3552:L P[2314]  R[157] mm/sec CNT100 Offset,PR[24:Rotate_Offset] ;
3553:L P[2315]  R[157] mm/sec CNT100 Offset,PR[24:Rotate_Offset] ;
3554:L P[2316]  R[157] mm/sec CNT100 Offset,PR[24:Rotate_Offset] ;
3555:L P[2317]  R[157] mm/sec CNT100 Offset,PR[24:Rotate_Offset] ;
3556: !Pass176 ;
3557: LBL[1176:Pass176] ;
3558:L P[2318]  R[157] mm/sec FINE Offset,PR[78:Offst_apprch]  ;
3559: WAIT   0.20(sec) ;
3560:L P[2318]  R[157] mm/sec CNT100 TA    0.00sec,CALL RUN_LASER_START Offset,PR[25:Start_Offset] ;
3562:L P[2319]  R[157] mm/sec CNT100 Offset,PR[24:Rotate_Offset] ;
3563:L P[2320]  R[157] mm/sec CNT100 Offset,PR[24:Rotate_Offset] ;
3564:L P[2321]  R[157] mm/sec CNT100 Offset,PR[24:Rotate_Offset] ;
3565:L P[2322]  R[157] mm/sec CNT100 TA    0.00sec,CALL RUN_LASER_STOP Offset,PR[26:Stop_Offset] ;
3567:L P[2322]  R[157] mm/sec FINE Offset,PR[76:Offst_dprt] ;
3568:L P[2323]  R[157] mm/sec CNT100 Offset,PR[24:Rotate_Offset] ;
3569:L P[2324]  R[157] mm/sec CNT100 Offset,PR[24:Rotate_Offset] ;
3570:L P[2325]  R[157] mm/sec CNT100 Offset,PR[24:Rotate_Offset] ;
3571:L P[2326]  R[157] mm/sec CNT100 Offset,PR[24:Rotate_Offset] ;
3572:L P[2327]  R[157] mm/sec CNT100 Offset,PR[24:Rotate_Offset] ;
3573:L P[2328]  R[157] mm/sec CNT100 Offset,PR[24:Rotate_Offset] ;
3574: !Pass177 ;
3575: LBL[1177:Pass177] ;
3576:L P[2329]  R[157] mm/sec FINE Offset,PR[78:Offst_apprch]  ;
3577: WAIT   0.20(sec) ;
3578:L P[2329]  R[157] mm/sec CNT100 TA    0.00sec,CALL RUN_LASER_START Offset,PR[25:Start_Offset] ;
3580:L P[2330]  R[157] mm/sec CNT100 Offset,PR[24:Rotate_Offset] ;
3581:L P[2331]  R[157] mm/sec CNT100 Offset,PR[24:Rotate_Offset] ;
3582:L P[2332]  R[157] mm/sec CNT100 Offset,PR[24:Rotate_Offset] ;
3583:L P[2333]  R[157] mm/sec CNT100 TA    0.00sec,CALL RUN_LASER_STOP Offset,PR[26:Stop_Offset] ;
3585:L P[2333]  R[157] mm/sec FINE Offset,PR[76:Offst_dprt] ;
3586:L P[2334]  R[157] mm/sec CNT100 Offset,PR[24:Rotate_Offset] ;
3587:L P[2335]  R[157] mm/sec CNT100 Offset,PR[24:Rotate_Offset] ;
3588:L P[2336]  R[157] mm/sec CNT100 Offset,PR[24:Rotate_Offset] ;
3589:L P[2337]  R[157] mm/sec CNT100 Offset,PR[24:Rotate_Offset] ;
3590:L P[2338]  R[157] mm/sec CNT100 Offset,PR[24:Rotate_Offset] ;
3591:L P[2339]  R[157] mm/sec CNT100 Offset,PR[24:Rotate_Offset] ;
3592: !Pass178 ;
3593: LBL[1178:Pass178] ;
3594:L P[2340]  R[157] mm/sec FINE Offset,PR[78:Offst_apprch]  ;
3595: WAIT   0.20(sec) ;
3596:L P[2340]  R[157] mm/sec CNT100 TA    0.00sec,CALL RUN_LASER_START Offset,PR[25:Start_Offset] ;
3598:L P[2341]  R[157] mm/sec CNT100 Offset,PR[24:Rotate_Offset] ;
3599:L P[2342]  R[157] mm/sec CNT100 Offset,PR[24:Rotate_Offset] ;
3600:L P[2343]  R[157] mm/sec CNT100 Offset,PR[24:Rotate_Offset] ;
3601:L P[2344]  R[157] mm/sec CNT100 TA    0.00sec,CALL RUN_LASER_STOP Offset,PR[26:Stop_Offset] ;
3603:L P[2344]  R[157] mm/sec FINE Offset,PR[76:Offst_dprt] ;
3604:L P[2345]  R[157] mm/sec CNT100 Offset,PR[24:Rotate_Offset] ;
3605:L P[2346]  R[157] mm/sec CNT100 Offset,PR[24:Rotate_Offset] ;
3606:L P[2347]  R[157] mm/sec CNT100 Offset,PR[24:Rotate_Offset] ;
3607:L P[2348]  R[157] mm/sec CNT100 Offset,PR[24:Rotate_Offset] ;
3608:L P[2349]  R[157] mm/sec CNT100 Offset,PR[24:Rotate_Offset] ;
3609:L P[2350]  R[157] mm/sec CNT100 Offset,PR[24:Rotate_Offset] ;
3610: !Pass179 ;
3611: LBL[1179:Pass179] ;
3612:L P[2351]  R[157] mm/sec FINE Offset,PR[78:Offst_apprch]  ;
3613: WAIT   0.20(sec) ;
3614:L P[2351]  R[157] mm/sec CNT100 TA    0.00sec,CALL RUN_LASER_START Offset,PR[25:Start_Offset] ;
3616:L P[2352]  R[157] mm/sec CNT100 Offset,PR[24:Rotate_Offset] ;
3617:L P[2353]  R[157] mm/sec CNT100 TA    0.00sec,CALL RUN_LASER_STOP Offset,PR[26:Stop_Offset] ;
3619:L P[2353]  R[157] mm/sec FINE Offset,PR[76:Offst_dprt] ;
3620:L P[2354]  R[157] mm/sec CNT100 Offset,PR[24:Rotate_Offset] ;
3621:L P[2355]  R[157] mm/sec CNT100 Offset,PR[24:Rotate_Offset] ;
3622:L P[2356]  R[157] mm/sec CNT100 Offset,PR[24:Rotate_Offset] ;
3623:L P[2357]  R[157] mm/sec CNT100 Offset,PR[24:Rotate_Offset] ;
3624:L P[2358]  R[157] mm/sec CNT100 Offset,PR[24:Rotate_Offset] ;
3625:L P[2359]  R[157] mm/sec CNT100 Offset,PR[24:Rotate_Offset] ;
3626: !Pass180 ;
3627: LBL[1180:Pass180] ;
3628:L P[2360]  R[157] mm/sec FINE Offset,PR[78:Offst_apprch]  ;
3629: WAIT   0.20(sec) ;
3630:L P[2360]  R[157] mm/sec CNT100 TA    0.00sec,CALL RUN_LASER_START Offset,PR[25:Start_Offset] ;
3632:L P[2361]  R[157] mm/sec CNT100 Offset,PR[24:Rotate_Offset] ;
3633:L P[2362]  R[157] mm/sec CNT100 TA    0.00sec,CALL RUN_LASER_STOP Offset,PR[26:Stop_Offset] ;
3635:L P[2362]  R[157] mm/sec FINE Offset,PR[76:Offst_dprt] ;
3636:L P[2363]  R[157] mm/sec CNT100 Offset,PR[24:Rotate_Offset] ;
3637:L P[2364]  R[157] mm/sec CNT100 Offset,PR[24:Rotate_Offset] ;
3638:L P[2365]  R[157] mm/sec CNT100 Offset,PR[24:Rotate_Offset] ;
3639:L P[2366]  R[157] mm/sec CNT100 Offset,PR[24:Rotate_Offset] ;
3640:L P[2367]  R[157] mm/sec CNT100 Offset,PR[24:Rotate_Offset] ;
3641:L P[2368]  R[157] mm/sec CNT100 Offset,PR[24:Rotate_Offset] ;
3642: !Pass181 ;
3643: LBL[1181:Pass181] ;
3644:L P[2369]  R[157] mm/sec FINE Offset,PR[78:Offst_apprch]  ;
3645: WAIT   0.20(sec) ;
3646:L P[2369]  R[157] mm/sec CNT100 TA    0.00sec,CALL RUN_LASER_START Offset,PR[25:Start_Offset] ;
3648:L P[2370]  R[157] mm/sec CNT100 Offset,PR[24:Rotate_Offset] ;
3649:L P[2371]  R[157] mm/sec CNT100 Offset,PR[24:Rotate_Offset] ;
3650:L P[2372]  R[157] mm/sec CNT100 Offset,PR[24:Rotate_Offset] ;
3651:L P[2373]  R[157] mm/sec CNT100 TA    0.00sec,CALL RUN_LASER_STOP Offset,PR[26:Stop_Offset] ;
3653:L P[2373]  R[157] mm/sec FINE Offset,PR[76:Offst_dprt] ;
3654:L P[2374]  R[157] mm/sec CNT100 Offset,PR[24:Rotate_Offset] ;
3655:L P[2375]  R[157] mm/sec CNT100 Offset,PR[24:Rotate_Offset] ;
3656:L P[2376]  R[157] mm/sec CNT100 Offset,PR[24:Rotate_Offset] ;
3657:L P[2377]  R[157] mm/sec CNT100 Offset,PR[24:Rotate_Offset] ;
3658:L P[2378]  R[157] mm/sec CNT100 Offset,PR[24:Rotate_Offset] ;
3659:L P[2379]  R[157] mm/sec CNT100 Offset,PR[24:Rotate_Offset] ;
3660: !Pass182 ;
3661: LBL[1182:Pass182] ;
3662:L P[2380]  R[157] mm/sec FINE Offset,PR[78:Offst_apprch]  ;
3663: WAIT   0.20(sec) ;
3664:L P[2380]  R[157] mm/sec CNT100 TA    0.00sec,CALL RUN_LASER_START Offset,PR[25:Start_Offset] ;
3666:L P[2381]  R[157] mm/sec CNT100 Offset,PR[24:Rotate_Offset] ;
3667:L P[2382]  R[157] mm/sec CNT100 Offset,PR[24:Rotate_Offset] ;
3668:L P[2383]  R[157] mm/sec CNT100 Offset,PR[24:Rotate_Offset] ;
3669:L P[2384]  R[157] mm/sec CNT100 TA    0.00sec,CALL RUN_LASER_STOP Offset,PR[26:Stop_Offset] ;
3671:L P[2384]  R[157] mm/sec FINE Offset,PR[76:Offst_dprt] ;
3672:L P[2385]  R[157] mm/sec CNT100 Offset,PR[24:Rotate_Offset] ;
3673:L P[2386]  R[157] mm/sec CNT100 Offset,PR[24:Rotate_Offset] ;
3674:L P[2387]  R[157] mm/sec CNT100 Offset,PR[24:Rotate_Offset] ;
3675:L P[2388]  R[157] mm/sec CNT100 Offset,PR[24:Rotate_Offset] ;
3676:L P[2389]  R[157] mm/sec CNT100 Offset,PR[24:Rotate_Offset] ;
3677:L P[2390]  R[157] mm/sec CNT100 Offset,PR[24:Rotate_Offset] ;
3678: !Pass183 ;
3679: LBL[1183:Pass183] ;
3680:L P[2391]  R[157] mm/sec FINE Offset,PR[78:Offst_apprch]  ;
3681: WAIT   0.20(sec) ;
3682:L P[2391]  R[157] mm/sec CNT100 TA    0.00sec,CALL RUN_LASER_START Offset,PR[25:Start_Offset] ;
3684:L P[2392]  R[157] mm/sec CNT100 Offset,PR[24:Rotate_Offset] ;
3685:L P[2393]  R[157] mm/sec CNT100 Offset,PR[24:Rotate_Offset] ;
3686:L P[2394]  R[157] mm/sec CNT100 Offset,PR[24:Rotate_Offset] ;
3687:L P[2395]  R[157] mm/sec CNT100 TA    0.00sec,CALL RUN_LASER_STOP Offset,PR[26:Stop_Offset] ;
3689:L P[2395]  R[157] mm/sec FINE Offset,PR[76:Offst_dprt] ;
3690:L P[2396]  R[157] mm/sec CNT100 Offset,PR[24:Rotate_Offset] ;
3691:L P[2397]  R[157] mm/sec CNT100 Offset,PR[24:Rotate_Offset] ;
3692:L P[2398]  R[157] mm/sec CNT100 Offset,PR[24:Rotate_Offset] ;
3693:L P[2399]  R[157] mm/sec CNT100 Offset,PR[24:Rotate_Offset] ;
3694:L P[2400]  R[157] mm/sec CNT100 Offset,PR[24:Rotate_Offset] ;
3695:L P[2401]  R[157] mm/sec CNT100 Offset,PR[24:Rotate_Offset] ;
3696: !Pass184 ;
3697: LBL[1184:Pass184] ;
3698:L P[2402]  R[157] mm/sec FINE Offset,PR[78:Offst_apprch]  ;
3699: WAIT   0.20(sec) ;
3700:L P[2402]  R[157] mm/sec CNT100 TA    0.00sec,CALL RUN_LASER_START Offset,PR[25:Start_Offset] ;
3702:L P[2403]  R[157] mm/sec CNT100 Offset,PR[24:Rotate_Offset] ;
3703:L P[2404]  R[157] mm/sec CNT100 Offset,PR[24:Rotate_Offset] ;
3704:L P[2405]  R[157] mm/sec CNT100 Offset,PR[24:Rotate_Offset] ;
3705:L P[2406]  R[157] mm/sec CNT100 TA    0.00sec,CALL RUN_LASER_STOP Offset,PR[26:Stop_Offset] ;
3707:L P[2406]  R[157] mm/sec FINE Offset,PR[76:Offst_dprt] ;
3708:L P[2407]  R[157] mm/sec CNT100 Offset,PR[24:Rotate_Offset] ;
3709:L P[2408]  R[157] mm/sec CNT100 Offset,PR[24:Rotate_Offset] ;
3710:L P[2409]  R[157] mm/sec CNT100 Offset,PR[24:Rotate_Offset] ;
3711:L P[2410]  R[157] mm/sec CNT100 Offset,PR[24:Rotate_Offset] ;
3712:L P[2411]  R[157] mm/sec CNT100 Offset,PR[24:Rotate_Offset] ;
3713:L P[2412]  R[157] mm/sec CNT100 Offset,PR[24:Rotate_Offset] ;
3714: !Pass185 ;
3715: LBL[1185:Pass185] ;
3716:L P[2413]  R[157] mm/sec FINE Offset,PR[78:Offst_apprch]  ;
3717: WAIT   0.20(sec) ;
3718:L P[2413]  R[157] mm/sec CNT100 TA    0.00sec,CALL RUN_LASER_START Offset,PR[25:Start_Offset] ;
3720:L P[2414]  R[157] mm/sec CNT100 Offset,PR[24:Rotate_Offset] ;
3721:L P[2415]  R[157] mm/sec CNT100 Offset,PR[24:Rotate_Offset] ;
3722:L P[2416]  R[157] mm/sec CNT100 Offset,PR[24:Rotate_Offset] ;
3723:L P[2417]  R[157] mm/sec CNT100 TA    0.00sec,CALL RUN_LASER_STOP Offset,PR[26:Stop_Offset] ;
3725:L P[2417]  R[157] mm/sec FINE Offset,PR[76:Offst_dprt] ;
3726:L P[2418]  R[157] mm/sec CNT100 Offset,PR[24:Rotate_Offset] ;
3727:L P[2419]  R[157] mm/sec CNT100 Offset,PR[24:Rotate_Offset] ;
3728:L P[2420]  R[157] mm/sec CNT100 Offset,PR[24:Rotate_Offset] ;
3729:L P[2421]  R[157] mm/sec CNT100 Offset,PR[24:Rotate_Offset] ;
3730:L P[2422]  R[157] mm/sec CNT100 Offset,PR[24:Rotate_Offset] ;
3731:L P[2423]  R[157] mm/sec CNT100 Offset,PR[24:Rotate_Offset] ;
3732: !Pass186 ;
3733: LBL[1186:Pass186] ;
3734:L P[2424]  R[157] mm/sec FINE Offset,PR[78:Offst_apprch]  ;
3735: WAIT   0.20(sec) ;
3736:L P[2424]  R[157] mm/sec CNT100 TA    0.00sec,CALL RUN_LASER_START Offset,PR[25:Start_Offset] ;
3738:L P[2425]  R[157] mm/sec CNT100 Offset,PR[24:Rotate_Offset] ;
3739:L P[2426]  R[157] mm/sec CNT100 Offset,PR[24:Rotate_Offset] ;
3740:L P[2427]  R[157] mm/sec CNT100 Offset,PR[24:Rotate_Offset] ;
3741:L P[2428]  R[157] mm/sec CNT100 Offset,PR[24:Rotate_Offset] ;
3742:L P[2429]  R[157] mm/sec CNT100 TA    0.00sec,CALL RUN_LASER_STOP Offset,PR[26:Stop_Offset] ;
3744:L P[2429]  R[157] mm/sec FINE Offset,PR[76:Offst_dprt] ;
3745:L P[2430]  R[157] mm/sec CNT100 Offset,PR[24:Rotate_Offset] ;
3746:L P[2431]  R[157] mm/sec CNT100 Offset,PR[24:Rotate_Offset] ;
3747:L P[2432]  R[157] mm/sec CNT100 Offset,PR[24:Rotate_Offset] ;
3748:L P[2433]  R[157] mm/sec CNT100 Offset,PR[24:Rotate_Offset] ;
3749:L P[2434]  R[157] mm/sec CNT100 Offset,PR[24:Rotate_Offset] ;
3750:L P[2435]  R[157] mm/sec CNT100 Offset,PR[24:Rotate_Offset] ;
3751: !Pass187 ;
3752: LBL[1187:Pass187] ;
3753:L P[2436]  R[157] mm/sec FINE Offset,PR[78:Offst_apprch]  ;
3754: WAIT   0.20(sec) ;
3755:L P[2436]  R[157] mm/sec CNT100 TA    0.00sec,CALL RUN_LASER_START Offset,PR[25:Start_Offset] ;
3757:L P[2437]  R[157] mm/sec CNT100 Offset,PR[24:Rotate_Offset] ;
3758:L P[2438]  R[157] mm/sec CNT100 TA    0.00sec,CALL RUN_LASER_STOP Offset,PR[26:Stop_Offset] ;
3760:L P[2438]  R[157] mm/sec FINE Offset,PR[76:Offst_dprt] ;
3761:L P[2439]  R[157] mm/sec CNT100 Offset,PR[24:Rotate_Offset] ;
3762:L P[2440]  R[157] mm/sec CNT100 Offset,PR[24:Rotate_Offset] ;
3763:L P[2441]  R[157] mm/sec CNT100 Offset,PR[24:Rotate_Offset] ;
3764:L P[2442]  R[157] mm/sec CNT100 Offset,PR[24:Rotate_Offset] ;
3765:L P[2443]  R[157] mm/sec CNT100 Offset,PR[24:Rotate_Offset] ;
3766:L P[2444]  R[157] mm/sec CNT100 Offset,PR[24:Rotate_Offset] ;
3767: !Pass188 ;
3768: LBL[1188:Pass188] ;
3769:L P[2445]  R[157] mm/sec FINE Offset,PR[78:Offst_apprch]  ;
3770: WAIT   0.20(sec) ;
3771:L P[2445]  R[157] mm/sec CNT100 TA    0.00sec,CALL RUN_LASER_START Offset,PR[25:Start_Offset] ;
3773:L P[2446]  R[157] mm/sec CNT100 Offset,PR[24:Rotate_Offset] ;
3774:L P[2447]  R[157] mm/sec CNT100 TA    0.00sec,CALL RUN_LASER_STOP Offset,PR[26:Stop_Offset] ;
3776:L P[2447]  R[157] mm/sec FINE Offset,PR[76:Offst_dprt] ;
3777:L P[2448]  R[157] mm/sec CNT100 Offset,PR[24:Rotate_Offset] ;
3778:L P[2449]  R[157] mm/sec CNT100 Offset,PR[24:Rotate_Offset] ;
3779:L P[2450]  R[157] mm/sec CNT100 Offset,PR[24:Rotate_Offset] ;
3780:L P[2451]  R[157] mm/sec CNT100 Offset,PR[24:Rotate_Offset] ;
3781:L P[2452]  R[157] mm/sec CNT100 Offset,PR[24:Rotate_Offset] ;
3782:L P[2453]  R[157] mm/sec CNT100 Offset,PR[24:Rotate_Offset] ;
3783: !Pass189 ;
3784: LBL[1189:Pass189] ;
3785:L P[2454]  R[157] mm/sec FINE Offset,PR[78:Offst_apprch]  ;
3786: WAIT   0.20(sec) ;
3787:L P[2454]  R[157] mm/sec CNT100 TA    0.00sec,CALL RUN_LASER_START Offset,PR[25:Start_Offset] ;
3789:L P[2455]  R[157] mm/sec CNT100 Offset,PR[24:Rotate_Offset] ;
3790:L P[2456]  R[157] mm/sec CNT100 Offset,PR[24:Rotate_Offset] ;
3791:L P[2457]  R[157] mm/sec CNT100 Offset,PR[24:Rotate_Offset] ;
3792:L P[2458]  R[157] mm/sec CNT100 Offset,PR[24:Rotate_Offset] ;
3793:L P[2459]  R[157] mm/sec CNT100 TA    0.00sec,CALL RUN_LASER_STOP Offset,PR[26:Stop_Offset] ;
3795:L P[2459]  R[157] mm/sec FINE Offset,PR[76:Offst_dprt] ;
3796:L P[2460]  R[157] mm/sec CNT100 Offset,PR[24:Rotate_Offset] ;
3797:L P[2461]  R[157] mm/sec CNT100 Offset,PR[24:Rotate_Offset] ;
3798:L P[2462]  R[157] mm/sec CNT100 Offset,PR[24:Rotate_Offset] ;
3799:L P[2463]  R[157] mm/sec CNT100 Offset,PR[24:Rotate_Offset] ;
3800:L P[2464]  R[157] mm/sec CNT100 Offset,PR[24:Rotate_Offset] ;
3801:L P[2465]  R[157] mm/sec CNT100 Offset,PR[24:Rotate_Offset] ;
3802: !Pass190 ;
3803: LBL[1190:Pass190] ;
3804:L P[2466]  R[157] mm/sec FINE Offset,PR[78:Offst_apprch]  ;
3805: WAIT   0.20(sec) ;
3806:L P[2466]  R[157] mm/sec CNT100 TA    0.00sec,CALL RUN_LASER_START Offset,PR[25:Start_Offset] ;
3808:L P[2467]  R[157] mm/sec CNT100 Offset,PR[24:Rotate_Offset] ;
3809:L P[2468]  R[157] mm/sec CNT100 Offset,PR[24:Rotate_Offset] ;
3810:L P[2469]  R[157] mm/sec CNT100 Offset,PR[24:Rotate_Offset] ;
3811:L P[2470]  R[157] mm/sec CNT100 TA    0.00sec,CALL RUN_LASER_STOP Offset,PR[26:Stop_Offset] ;
3813:L P[2470]  R[157] mm/sec FINE Offset,PR[76:Offst_dprt] ;
3814:L P[2471]  R[157] mm/sec CNT100 Offset,PR[24:Rotate_Offset] ;
3815:L P[2472]  R[157] mm/sec CNT100 Offset,PR[24:Rotate_Offset] ;
3816:L P[2473]  R[157] mm/sec CNT100 Offset,PR[24:Rotate_Offset] ;
3817:L P[2474]  R[157] mm/sec CNT100 Offset,PR[24:Rotate_Offset] ;
3818:L P[2475]  R[157] mm/sec CNT100 Offset,PR[24:Rotate_Offset] ;
3819:L P[2476]  R[157] mm/sec CNT100 Offset,PR[24:Rotate_Offset] ;
3820: !Pass191 ;
3821: LBL[1191:Pass191] ;
3822:L P[2477]  R[157] mm/sec FINE Offset,PR[78:Offst_apprch]  ;
3823: WAIT   0.20(sec) ;
3824:L P[2477]  R[157] mm/sec CNT100 TA    0.00sec,CALL RUN_LASER_START Offset,PR[25:Start_Offset] ;
3826:L P[2478]  R[157] mm/sec CNT100 Offset,PR[24:Rotate_Offset] ;
3827:L P[2479]  R[157] mm/sec CNT100 Offset,PR[24:Rotate_Offset] ;
3828:L P[2480]  R[157] mm/sec CNT100 Offset,PR[24:Rotate_Offset] ;
3829:L P[2481]  R[157] mm/sec CNT100 TA    0.00sec,CALL RUN_LASER_STOP Offset,PR[26:Stop_Offset] ;
3831:L P[2481]  R[157] mm/sec FINE Offset,PR[76:Offst_dprt] ;
3832:L P[2482]  R[157] mm/sec CNT100 Offset,PR[24:Rotate_Offset] ;
3833:L P[2483]  R[157] mm/sec CNT100 Offset,PR[24:Rotate_Offset] ;
3834:L P[2484]  R[157] mm/sec CNT100 Offset,PR[24:Rotate_Offset] ;
3835:L P[2485]  R[157] mm/sec CNT100 Offset,PR[24:Rotate_Offset] ;
3836:L P[2486]  R[157] mm/sec CNT100 Offset,PR[24:Rotate_Offset] ;
3837:L P[2487]  R[157] mm/sec CNT100 Offset,PR[24:Rotate_Offset] ;
3838: !Pass192 ;
3839: LBL[1192:Pass192] ;
3840:L P[2488]  R[157] mm/sec FINE Offset,PR[78:Offst_apprch]  ;
3841: WAIT   0.20(sec) ;
3842:L P[2488]  R[157] mm/sec CNT100 TA    0.00sec,CALL RUN_LASER_START Offset,PR[25:Start_Offset] ;
3844:L P[2489]  R[157] mm/sec CNT100 Offset,PR[24:Rotate_Offset] ;
3845:L P[2490]  R[157] mm/sec CNT100 Offset,PR[24:Rotate_Offset] ;
3846:L P[2491]  R[157] mm/sec CNT100 Offset,PR[24:Rotate_Offset] ;
3847:L P[2492]  R[157] mm/sec CNT100 TA    0.00sec,CALL RUN_LASER_STOP Offset,PR[26:Stop_Offset] ;
3849:L P[2492]  R[157] mm/sec FINE Offset,PR[76:Offst_dprt] ;
3850:L P[2493]  R[157] mm/sec CNT100 Offset,PR[24:Rotate_Offset] ;
3851:L P[2494]  R[157] mm/sec CNT100 Offset,PR[24:Rotate_Offset] ;
3852:L P[2495]  R[157] mm/sec CNT100 Offset,PR[24:Rotate_Offset] ;
3853:L P[2496]  R[157] mm/sec CNT100 Offset,PR[24:Rotate_Offset] ;
3854:L P[2497]  R[157] mm/sec CNT100 Offset,PR[24:Rotate_Offset] ;
3855:L P[2498]  R[157] mm/sec CNT100 Offset,PR[24:Rotate_Offset] ;
3856: !Pass193 ;
3857: LBL[1193:Pass193] ;
3858:L P[2499]  R[157] mm/sec FINE Offset,PR[78:Offst_apprch]  ;
3859: WAIT   0.20(sec) ;
3860:L P[2499]  R[157] mm/sec CNT100 TA    0.00sec,CALL RUN_LASER_START Offset,PR[25:Start_Offset] ;
3862:L P[2500]  R[157] mm/sec CNT100 Offset,PR[24:Rotate_Offset] ;
3863:L P[2501]  R[157] mm/sec CNT100 Offset,PR[24:Rotate_Offset] ;
3864:L P[2502]  R[157] mm/sec CNT100 Offset,PR[24:Rotate_Offset] ;
3865:L P[2503]  R[157] mm/sec CNT100 TA    0.00sec,CALL RUN_LASER_STOP Offset,PR[26:Stop_Offset] ;
3867:L P[2503]  R[157] mm/sec FINE Offset,PR[76:Offst_dprt] ;
3868:L P[2504]  R[157] mm/sec CNT100 Offset,PR[24:Rotate_Offset] ;
3869:L P[2505]  R[157] mm/sec CNT100 Offset,PR[24:Rotate_Offset] ;
3870:L P[2506]  R[157] mm/sec CNT100 Offset,PR[24:Rotate_Offset] ;
3871:L P[2507]  R[157] mm/sec CNT100 Offset,PR[24:Rotate_Offset] ;
3872:L P[2508]  R[157] mm/sec CNT100 Offset,PR[24:Rotate_Offset] ;
3873:L P[2509]  R[157] mm/sec CNT100 Offset,PR[24:Rotate_Offset] ;
3874: !Pass194 ;
3875: LBL[1194:Pass194] ;
3876:L P[2510]  R[157] mm/sec FINE Offset,PR[78:Offst_apprch]  ;
3877: WAIT   0.20(sec) ;
3878:L P[2510]  R[157] mm/sec CNT100 TA    0.00sec,CALL RUN_LASER_START Offset,PR[25:Start_Offset] ;
3880:L P[2511]  R[157] mm/sec CNT100 Offset,PR[24:Rotate_Offset] ;
3881:L P[2512]  R[157] mm/sec CNT100 Offset,PR[24:Rotate_Offset] ;
3882:L P[2513]  R[157] mm/sec CNT100 Offset,PR[24:Rotate_Offset] ;
3883:L P[2514]  R[157] mm/sec CNT100 TA    0.00sec,CALL RUN_LASER_STOP Offset,PR[26:Stop_Offset] ;
3885:L P[2514]  R[157] mm/sec FINE Offset,PR[76:Offst_dprt] ;
3886:L P[2515]  R[157] mm/sec CNT100 Offset,PR[24:Rotate_Offset] ;
3887:L P[2516]  R[157] mm/sec CNT100 Offset,PR[24:Rotate_Offset] ;
3888:L P[2517]  R[157] mm/sec CNT100 Offset,PR[24:Rotate_Offset] ;
3889:L P[2518]  R[157] mm/sec CNT100 Offset,PR[24:Rotate_Offset] ;
3890:L P[2519]  R[157] mm/sec CNT100 Offset,PR[24:Rotate_Offset] ;
3891:L P[2520]  R[157] mm/sec CNT100 Offset,PR[24:Rotate_Offset] ;
3892: !Pass195 ;
3893: LBL[1195:Pass195] ;
3894:L P[2521]  R[157] mm/sec FINE Offset,PR[78:Offst_apprch]  ;
3895: WAIT   0.20(sec) ;
3896:L P[2521]  R[157] mm/sec CNT100 TA    0.00sec,CALL RUN_LASER_START Offset,PR[25:Start_Offset] ;
3898:L P[2522]  R[157] mm/sec CNT100 Offset,PR[24:Rotate_Offset] ;
3899:L P[2523]  R[157] mm/sec CNT100 TA    0.00sec,CALL RUN_LASER_STOP Offset,PR[26:Stop_Offset] ;
3901:L P[2523]  R[157] mm/sec FINE Offset,PR[76:Offst_dprt] ;
3902:L P[2524]  R[157] mm/sec CNT100 Offset,PR[24:Rotate_Offset] ;
3903:L P[2525]  R[157] mm/sec CNT100 Offset,PR[24:Rotate_Offset] ;
3904:L P[2526]  R[157] mm/sec CNT100 Offset,PR[24:Rotate_Offset] ;
3905:L P[2527]  R[157] mm/sec CNT100 Offset,PR[24:Rotate_Offset] ;
3906:L P[2528]  R[157] mm/sec CNT100 Offset,PR[24:Rotate_Offset] ;
3907:L P[2529]  R[157] mm/sec CNT100 Offset,PR[24:Rotate_Offset] ;
3908: !Pass196 ;
3909: LBL[1196:Pass196] ;
3910:L P[2530]  R[157] mm/sec FINE Offset,PR[78:Offst_apprch]  ;
3911: WAIT   0.20(sec) ;
3912:L P[2530]  R[157] mm/sec CNT100 TA    0.00sec,CALL RUN_LASER_START Offset,PR[25:Start_Offset] ;
3914:L P[2531]  R[157] mm/sec CNT100 Offset,PR[24:Rotate_Offset] ;
3915:L P[2532]  R[157] mm/sec CNT100 TA    0.00sec,CALL RUN_LASER_STOP Offset,PR[26:Stop_Offset] ;
3917:L P[2532]  R[157] mm/sec FINE Offset,PR[76:Offst_dprt] ;
3918:L P[2533]  R[157] mm/sec CNT100 Offset,PR[24:Rotate_Offset] ;
3919:L P[2534]  R[157] mm/sec CNT100 Offset,PR[24:Rotate_Offset] ;
3920:L P[2535]  R[157] mm/sec CNT100 Offset,PR[24:Rotate_Offset] ;
3921:L P[2536]  R[157] mm/sec CNT100 Offset,PR[24:Rotate_Offset] ;
3922:L P[2537]  R[157] mm/sec CNT100 Offset,PR[24:Rotate_Offset] ;
3923:L P[2538]  R[157] mm/sec CNT100 Offset,PR[24:Rotate_Offset] ;
3924: !Pass197 ;
3925: LBL[1197:Pass197] ;
3926:L P[2539]  R[157] mm/sec FINE Offset,PR[78:Offst_apprch]  ;
3927: WAIT   0.20(sec) ;
3928:L P[2539]  R[157] mm/sec CNT100 TA    0.00sec,CALL RUN_LASER_START Offset,PR[25:Start_Offset] ;
3930:L P[2540]  R[157] mm/sec CNT100 Offset,PR[24:Rotate_Offset] ;
3931:L P[2541]  R[157] mm/sec CNT100 Offset,PR[24:Rotate_Offset] ;
3932:L P[2542]  R[157] mm/sec CNT100 Offset,PR[24:Rotate_Offset] ;
3933:L P[2543]  R[157] mm/sec CNT100 TA    0.00sec,CALL RUN_LASER_STOP Offset,PR[26:Stop_Offset] ;
3935:L P[2543]  R[157] mm/sec FINE Offset,PR[76:Offst_dprt] ;
3936:L P[2544]  R[157] mm/sec CNT100 Offset,PR[24:Rotate_Offset] ;
3937:L P[2545]  R[157] mm/sec CNT100 Offset,PR[24:Rotate_Offset] ;
3938:L P[2546]  R[157] mm/sec CNT100 Offset,PR[24:Rotate_Offset] ;
3939:L P[2547]  R[157] mm/sec CNT100 Offset,PR[24:Rotate_Offset] ;
3940:L P[2548]  R[157] mm/sec CNT100 Offset,PR[24:Rotate_Offset] ;
3941:L P[2549]  R[157] mm/sec CNT100 Offset,PR[24:Rotate_Offset] ;
3942: !Pass198 ;
3943: LBL[1198:Pass198] ;
3944:L P[2550]  R[157] mm/sec FINE Offset,PR[78:Offst_apprch]  ;
3945: WAIT   0.20(sec) ;
3946:L P[2550]  R[157] mm/sec CNT100 TA    0.00sec,CALL RUN_LASER_START Offset,PR[25:Start_Offset] ;
3948:L P[2551]  R[157] mm/sec CNT100 Offset,PR[24:Rotate_Offset] ;
3949:L P[2552]  R[157] mm/sec CNT100 Offset,PR[24:Rotate_Offset] ;
3950:L P[2553]  R[157] mm/sec CNT100 Offset,PR[24:Rotate_Offset] ;
3951:L P[2554]  R[157] mm/sec CNT100 TA    0.00sec,CALL RUN_LASER_STOP Offset,PR[26:Stop_Offset] ;
3953:L P[2554]  R[157] mm/sec FINE Offset,PR[76:Offst_dprt] ;
3954:L P[2555]  R[157] mm/sec CNT100 Offset,PR[24:Rotate_Offset] ;
3955:L P[2556]  R[157] mm/sec CNT100 Offset,PR[24:Rotate_Offset] ;
3956:L P[2557]  R[157] mm/sec CNT100 Offset,PR[24:Rotate_Offset] ;
3957:L P[2558]  R[157] mm/sec CNT100 Offset,PR[24:Rotate_Offset] ;
3958:L P[2559]  R[157] mm/sec CNT100 Offset,PR[24:Rotate_Offset] ;
3959:L P[2560]  R[157] mm/sec CNT100 Offset,PR[24:Rotate_Offset] ;
3960: !Pass199 ;
3961: LBL[1199:Pass199] ;
3962:L P[2561]  R[157] mm/sec FINE Offset,PR[78:Offst_apprch]  ;
3963: WAIT   0.20(sec) ;
3964:L P[2561]  R[157] mm/sec CNT100 TA    0.00sec,CALL RUN_LASER_START Offset,PR[25:Start_Offset] ;
3966:L P[2562]  R[157] mm/sec CNT100 Offset,PR[24:Rotate_Offset] ;
3967:L P[2563]  R[157] mm/sec CNT100 Offset,PR[24:Rotate_Offset] ;
3968:L P[2564]  R[157] mm/sec CNT100 Offset,PR[24:Rotate_Offset] ;
3969:L P[2565]  R[157] mm/sec CNT100 TA    0.00sec,CALL RUN_LASER_STOP Offset,PR[26:Stop_Offset] ;
3971:L P[2565]  R[157] mm/sec FINE Offset,PR[76:Offst_dprt] ;
3972:L P[2566]  R[157] mm/sec CNT100 Offset,PR[24:Rotate_Offset] ;
3973:L P[2567]  R[157] mm/sec CNT100 Offset,PR[24:Rotate_Offset] ;
3974:L P[2568]  R[157] mm/sec CNT100 Offset,PR[24:Rotate_Offset] ;
3975:L P[2569]  R[157] mm/sec CNT100 Offset,PR[24:Rotate_Offset] ;
3976:L P[2570]  R[157] mm/sec CNT100 Offset,PR[24:Rotate_Offset] ;
3977:L P[2571]  R[157] mm/sec CNT100 Offset,PR[24:Rotate_Offset] ;
3978: !Pass200 ;
3979: LBL[1200:Pass200] ;
3980:L P[2572]  R[157] mm/sec FINE Offset,PR[78:Offst_apprch]  ;
3981: WAIT   0.20(sec) ;
3982:L P[2572]  R[157] mm/sec CNT100 TA    0.00sec,CALL RUN_LASER_START Offset,PR[25:Start_Offset] ;
3984:L P[2573]  R[157] mm/sec CNT100 Offset,PR[24:Rotate_Offset] ;
3985:L P[2574]  R[157] mm/sec CNT100 Offset,PR[24:Rotate_Offset] ;
3986:L P[2575]  R[157] mm/sec CNT100 Offset,PR[24:Rotate_Offset] ;
3987:L P[2576]  R[157] mm/sec CNT100 TA    0.00sec,CALL RUN_LASER_STOP Offset,PR[26:Stop_Offset] ;
3989:L P[2576]  R[157] mm/sec FINE Offset,PR[76:Offst_dprt] ;
3990:L P[2577]  R[157] mm/sec CNT100 Offset,PR[24:Rotate_Offset] ;
3991:L P[2578]  R[157] mm/sec CNT100 Offset,PR[24:Rotate_Offset] ;
3992:L P[2579]  R[157] mm/sec CNT100 Offset,PR[24:Rotate_Offset] ;
3993:L P[2580]  R[157] mm/sec CNT100 Offset,PR[24:Rotate_Offset] ;
3994:L P[2581]  R[157] mm/sec CNT100 Offset,PR[24:Rotate_Offset] ;
3995:L P[2582]  R[157] mm/sec CNT100 Offset,PR[24:Rotate_Offset] ;
3996: !Pass201 ;
3997: LBL[1201:Pass201] ;
3998:L P[2583]  R[157] mm/sec FINE Offset,PR[78:Offst_apprch]  ;
3999: WAIT   0.20(sec) ;
4000:L P[2583]  R[157] mm/sec CNT100 TA    0.00sec,CALL RUN_LASER_START Offset,PR[25:Start_Offset] ;
4002:L P[2584]  R[157] mm/sec CNT100 Offset,PR[24:Rotate_Offset] ;
4003:L P[2585]  R[157] mm/sec CNT100 Offset,PR[24:Rotate_Offset] ;
4004:L P[2586]  R[157] mm/sec CNT100 Offset,PR[24:Rotate_Offset] ;
4005:L P[2587]  R[157] mm/sec CNT100 TA    0.00sec,CALL RUN_LASER_STOP Offset,PR[26:Stop_Offset] ;
4007:L P[2587]  R[157] mm/sec FINE Offset,PR[76:Offst_dprt] ;
4008:L P[2588]  R[157] mm/sec CNT100 Offset,PR[24:Rotate_Offset] ;
4009:L P[2589]  R[157] mm/sec CNT100 Offset,PR[24:Rotate_Offset] ;
4010:L P[2590]  R[157] mm/sec CNT100 Offset,PR[24:Rotate_Offset] ;
4011:L P[2591]  R[157] mm/sec CNT100 Offset,PR[24:Rotate_Offset] ;
4012:L P[2592]  R[157] mm/sec CNT100 Offset,PR[24:Rotate_Offset] ;
4013:L P[2593]  R[157] mm/sec CNT100 Offset,PR[24:Rotate_Offset] ;
4014: !Pass202 ;
4015: LBL[1202:Pass202] ;
4016:L P[2594]  R[157] mm/sec FINE Offset,PR[78:Offst_apprch]  ;
4017: WAIT   0.20(sec) ;
4018:L P[2594]  R[157] mm/sec CNT100 TA    0.00sec,CALL RUN_LASER_START Offset,PR[25:Start_Offset] ;
4020:L P[2595]  R[157] mm/sec CNT100 Offset,PR[24:Rotate_Offset] ;
4021:L P[2596]  R[157] mm/sec CNT100 Offset,PR[24:Rotate_Offset] ;
4022:L P[2597]  R[157] mm/sec CNT100 Offset,PR[24:Rotate_Offset] ;
4023:L P[2598]  R[157] mm/sec CNT100 Offset,PR[24:Rotate_Offset] ;
4024:L P[2599]  R[157] mm/sec CNT100 TA    0.00sec,CALL RUN_LASER_STOP Offset,PR[26:Stop_Offset] ;
4026:L P[2599]  R[157] mm/sec FINE Offset,PR[76:Offst_dprt] ;
4027:L P[2600]  R[157] mm/sec CNT100 Offset,PR[24:Rotate_Offset] ;
4028:L P[2601]  R[157] mm/sec CNT100 Offset,PR[24:Rotate_Offset] ;
4029:L P[2602]  R[157] mm/sec CNT100 Offset,PR[24:Rotate_Offset] ;
4030:L P[2603]  R[157] mm/sec CNT100 Offset,PR[24:Rotate_Offset] ;
4031:L P[2604]  R[157] mm/sec CNT100 Offset,PR[24:Rotate_Offset] ;
4032:L P[2605]  R[157] mm/sec CNT100 Offset,PR[24:Rotate_Offset] ;
4033: !Pass203 ;
4034: LBL[1203:Pass203] ;
4035:L P[2606]  R[157] mm/sec FINE Offset,PR[78:Offst_apprch]  ;
4036: WAIT   0.20(sec) ;
4037:L P[2606]  R[157] mm/sec CNT100 TA    0.00sec,CALL RUN_LASER_START Offset,PR[25:Start_Offset] ;
4039:L P[2607]  R[157] mm/sec CNT100 Offset,PR[24:Rotate_Offset] ;
4040:L P[2608]  R[157] mm/sec CNT100 TA    0.00sec,CALL RUN_LASER_STOP Offset,PR[26:Stop_Offset] ;
4042:L P[2608]  R[157] mm/sec FINE Offset,PR[76:Offst_dprt] ;
4043:L P[2609]  R[157] mm/sec CNT100 Offset,PR[24:Rotate_Offset] ;
4044:L P[2610]  R[157] mm/sec CNT100 Offset,PR[24:Rotate_Offset] ;
4045:L P[2611]  R[157] mm/sec CNT100 Offset,PR[24:Rotate_Offset] ;
4046:L P[2612]  R[157] mm/sec CNT100 Offset,PR[24:Rotate_Offset] ;
4047:L P[2613]  R[157] mm/sec CNT100 Offset,PR[24:Rotate_Offset] ;
4048:L P[2614]  R[157] mm/sec CNT100 Offset,PR[24:Rotate_Offset] ;
4049: !Pass204 ;
4050: LBL[1204:Pass204] ;
4051:L P[2615]  R[157] mm/sec FINE Offset,PR[78:Offst_apprch]  ;
4052: WAIT   0.20(sec) ;
4053:L P[2615]  R[157] mm/sec CNT100 TA    0.00sec,CALL RUN_LASER_START Offset,PR[25:Start_Offset] ;
4055:L P[2616]  R[157] mm/sec CNT100 Offset,PR[24:Rotate_Offset] ;
4056:L P[2617]  R[157] mm/sec CNT100 TA    0.00sec,CALL RUN_LASER_STOP Offset,PR[26:Stop_Offset] ;
4058:L P[2617]  R[157] mm/sec FINE Offset,PR[76:Offst_dprt] ;
4059:L P[2618]  R[157] mm/sec CNT100 Offset,PR[24:Rotate_Offset] ;
4060:L P[2619]  R[157] mm/sec CNT100 Offset,PR[24:Rotate_Offset] ;
4061:L P[2620]  R[157] mm/sec CNT100 Offset,PR[24:Rotate_Offset] ;
4062:L P[2621]  R[157] mm/sec CNT100 Offset,PR[24:Rotate_Offset] ;
4063:L P[2622]  R[157] mm/sec CNT100 Offset,PR[24:Rotate_Offset] ;
4064:L P[2623]  R[157] mm/sec CNT100 Offset,PR[24:Rotate_Offset] ;
4065: !Pass205 ;
4066: LBL[1205:Pass205] ;
4067:L P[2624]  R[157] mm/sec FINE Offset,PR[78:Offst_apprch]  ;
4068: WAIT   0.20(sec) ;
4069:L P[2624]  R[157] mm/sec CNT100 TA    0.00sec,CALL RUN_LASER_START Offset,PR[25:Start_Offset] ;
4071:L P[2625]  R[157] mm/sec CNT100 Offset,PR[24:Rotate_Offset] ;
4072:L P[2626]  R[157] mm/sec CNT100 Offset,PR[24:Rotate_Offset] ;
4073:L P[2627]  R[157] mm/sec CNT100 Offset,PR[24:Rotate_Offset] ;
4074:L P[2628]  R[157] mm/sec CNT100 Offset,PR[24:Rotate_Offset] ;
4075:L P[2629]  R[157] mm/sec CNT100 TA    0.00sec,CALL RUN_LASER_STOP Offset,PR[26:Stop_Offset] ;
4077:L P[2629]  R[157] mm/sec FINE Offset,PR[76:Offst_dprt] ;
4078:L P[2630]  R[157] mm/sec CNT100 Offset,PR[24:Rotate_Offset] ;
4079:L P[2631]  R[157] mm/sec CNT100 Offset,PR[24:Rotate_Offset] ;
4080:L P[2632]  R[157] mm/sec CNT100 Offset,PR[24:Rotate_Offset] ;
4081:L P[2633]  R[157] mm/sec CNT100 Offset,PR[24:Rotate_Offset] ;
4082:L P[2634]  R[157] mm/sec CNT100 Offset,PR[24:Rotate_Offset] ;
4083:L P[2635]  R[157] mm/sec CNT100 Offset,PR[24:Rotate_Offset] ;
4084: !Pass206 ;
4085: LBL[1206:Pass206] ;
4086:L P[2636]  R[157] mm/sec FINE Offset,PR[78:Offst_apprch]  ;
4087: WAIT   0.20(sec) ;
4088:L P[2636]  R[157] mm/sec CNT100 TA    0.00sec,CALL RUN_LASER_START Offset,PR[25:Start_Offset] ;
4090:L P[2637]  R[157] mm/sec CNT100 Offset,PR[24:Rotate_Offset] ;
4091:L P[2638]  R[157] mm/sec CNT100 Offset,PR[24:Rotate_Offset] ;
4092:L P[2639]  R[157] mm/sec CNT100 Offset,PR[24:Rotate_Offset] ;
4093:L P[2640]  R[157] mm/sec CNT100 Offset,PR[24:Rotate_Offset] ;
4094:L P[2641]  R[157] mm/sec CNT100 TA    0.00sec,CALL RUN_LASER_STOP Offset,PR[26:Stop_Offset] ;
4096:L P[2641]  R[157] mm/sec FINE Offset,PR[76:Offst_dprt] ;
4097:L P[2642]  R[157] mm/sec CNT100 Offset,PR[24:Rotate_Offset] ;
4098:L P[2643]  R[157] mm/sec CNT100 Offset,PR[24:Rotate_Offset] ;
4099:L P[2644]  R[157] mm/sec CNT100 Offset,PR[24:Rotate_Offset] ;
4100:L P[2645]  R[157] mm/sec CNT100 Offset,PR[24:Rotate_Offset] ;
4101:L P[2646]  R[157] mm/sec CNT100 Offset,PR[24:Rotate_Offset] ;
4102:L P[2647]  R[157] mm/sec CNT100 Offset,PR[24:Rotate_Offset] ;
4103: !Pass207 ;
4104: LBL[1207:Pass207] ;
4105:L P[2648]  R[157] mm/sec FINE Offset,PR[78:Offst_apprch]  ;
4106: WAIT   0.20(sec) ;
4107:L P[2648]  R[157] mm/sec CNT100 TA    0.00sec,CALL RUN_LASER_START Offset,PR[25:Start_Offset] ;
4109:L P[2649]  R[157] mm/sec CNT100 Offset,PR[24:Rotate_Offset] ;
4110:L P[2650]  R[157] mm/sec CNT100 Offset,PR[24:Rotate_Offset] ;
4111:L P[2651]  R[157] mm/sec CNT100 Offset,PR[24:Rotate_Offset] ;
4112:L P[2652]  R[157] mm/sec CNT100 TA    0.00sec,CALL RUN_LASER_STOP Offset,PR[26:Stop_Offset] ;
4114:L P[2652]  R[157] mm/sec FINE Offset,PR[76:Offst_dprt] ;
4115:L P[2653]  R[157] mm/sec CNT100 Offset,PR[24:Rotate_Offset] ;
4116:L P[2654]  R[157] mm/sec CNT100 Offset,PR[24:Rotate_Offset] ;
4117:L P[2655]  R[157] mm/sec CNT100 Offset,PR[24:Rotate_Offset] ;
4118:L P[2656]  R[157] mm/sec CNT100 Offset,PR[24:Rotate_Offset] ;
4119:L P[2657]  R[157] mm/sec CNT100 Offset,PR[24:Rotate_Offset] ;
4120:L P[2658]  R[157] mm/sec CNT100 Offset,PR[24:Rotate_Offset] ;
4121: !Pass208 ;
4122: LBL[1208:Pass208] ;
4123:L P[2659]  R[157] mm/sec FINE Offset,PR[78:Offst_apprch]  ;
4124: WAIT   0.20(sec) ;
4125:L P[2659]  R[157] mm/sec CNT100 TA    0.00sec,CALL RUN_LASER_START Offset,PR[25:Start_Offset] ;
4127:L P[2660]  R[157] mm/sec CNT100 Offset,PR[24:Rotate_Offset] ;
4128:L P[2661]  R[157] mm/sec CNT100 Offset,PR[24:Rotate_Offset] ;
4129:L P[2662]  R[157] mm/sec CNT100 Offset,PR[24:Rotate_Offset] ;
4130:L P[2663]  R[157] mm/sec CNT100 TA    0.00sec,CALL RUN_LASER_STOP Offset,PR[26:Stop_Offset] ;
4132:L P[2663]  R[157] mm/sec FINE Offset,PR[76:Offst_dprt] ;
4133:L P[2664]  R[157] mm/sec CNT100 Offset,PR[24:Rotate_Offset] ;
4134:L P[2665]  R[157] mm/sec CNT100 Offset,PR[24:Rotate_Offset] ;
4135:L P[2666]  R[157] mm/sec CNT100 Offset,PR[24:Rotate_Offset] ;
4136:L P[2667]  R[157] mm/sec CNT100 Offset,PR[24:Rotate_Offset] ;
4137:L P[2668]  R[157] mm/sec CNT100 Offset,PR[24:Rotate_Offset] ;
4138:L P[2669]  R[157] mm/sec CNT100 Offset,PR[24:Rotate_Offset] ;
4139: !Pass209 ;
4140: LBL[1209:Pass209] ;
4141:L P[2670]  R[157] mm/sec FINE Offset,PR[78:Offst_apprch]  ;
4142: WAIT   0.20(sec) ;
4143:L P[2670]  R[157] mm/sec CNT100 TA    0.00sec,CALL RUN_LASER_START Offset,PR[25:Start_Offset] ;
4145:L P[2671]  R[157] mm/sec CNT100 Offset,PR[24:Rotate_Offset] ;
4146:L P[2672]  R[157] mm/sec CNT100 Offset,PR[24:Rotate_Offset] ;
4147:L P[2673]  R[157] mm/sec CNT100 Offset,PR[24:Rotate_Offset] ;
4148:L P[2674]  R[157] mm/sec CNT100 TA    0.00sec,CALL RUN_LASER_STOP Offset,PR[26:Stop_Offset] ;
4150:L P[2674]  R[157] mm/sec FINE Offset,PR[76:Offst_dprt] ;
4151:L P[2675]  R[157] mm/sec CNT100 Offset,PR[24:Rotate_Offset] ;
4152:L P[2676]  R[157] mm/sec CNT100 Offset,PR[24:Rotate_Offset] ;
4153:L P[2677]  R[157] mm/sec CNT100 Offset,PR[24:Rotate_Offset] ;
4154:L P[2678]  R[157] mm/sec CNT100 Offset,PR[24:Rotate_Offset] ;
4155:L P[2679]  R[157] mm/sec CNT100 Offset,PR[24:Rotate_Offset] ;
4156:L P[2680]  R[157] mm/sec CNT100 Offset,PR[24:Rotate_Offset] ;
4157: !Pass210 ;
4158: LBL[1210:Pass210] ;
4159:L P[2681]  R[157] mm/sec FINE Offset,PR[78:Offst_apprch]  ;
4160: WAIT   0.20(sec) ;
4161:L P[2681]  R[157] mm/sec CNT100 TA    0.00sec,CALL RUN_LASER_START Offset,PR[25:Start_Offset] ;
4163:L P[2682]  R[157] mm/sec CNT100 Offset,PR[24:Rotate_Offset] ;
4164:L P[2683]  R[157] mm/sec CNT100 Offset,PR[24:Rotate_Offset] ;
4165:L P[2684]  R[157] mm/sec CNT100 Offset,PR[24:Rotate_Offset] ;
4166:L P[2685]  R[157] mm/sec CNT100 TA    0.00sec,CALL RUN_LASER_STOP Offset,PR[26:Stop_Offset] ;
4168:L P[2685]  R[157] mm/sec FINE Offset,PR[76:Offst_dprt] ;
4169:L P[2686]  R[157] mm/sec CNT100 Offset,PR[24:Rotate_Offset] ;
4170:L P[2687]  R[157] mm/sec CNT100 Offset,PR[24:Rotate_Offset] ;
4171:L P[2688]  R[157] mm/sec CNT100 Offset,PR[24:Rotate_Offset] ;
4172:L P[2689]  R[157] mm/sec CNT100 Offset,PR[24:Rotate_Offset] ;
4173:L P[2690]  R[157] mm/sec CNT100 Offset,PR[24:Rotate_Offset] ;
4174:L P[2691]  R[157] mm/sec CNT100 Offset,PR[24:Rotate_Offset] ;
4175: !Pass211 ;
4176: LBL[1211:Pass211] ;
4177:L P[2692]  R[157] mm/sec FINE Offset,PR[78:Offst_apprch]  ;
4178: WAIT   0.20(sec) ;
4179:L P[2692]  R[157] mm/sec CNT100 TA    0.00sec,CALL RUN_LASER_START Offset,PR[25:Start_Offset] ;
4181:L P[2693]  R[157] mm/sec CNT100 Offset,PR[24:Rotate_Offset] ;
4182:L P[2694]  R[157] mm/sec CNT100 TA    0.00sec,CALL RUN_LASER_STOP Offset,PR[26:Stop_Offset] ;
4184:L P[2694]  R[157] mm/sec FINE Offset,PR[76:Offst_dprt] ;
4185:L P[2695]  R[157] mm/sec CNT100 Offset,PR[24:Rotate_Offset] ;
4186:L P[2696]  R[157] mm/sec CNT100 Offset,PR[24:Rotate_Offset] ;
4187:L P[2697]  R[157] mm/sec CNT100 Offset,PR[24:Rotate_Offset] ;
4188:L P[2698]  R[157] mm/sec CNT100 Offset,PR[24:Rotate_Offset] ;
4189:L P[2699]  R[157] mm/sec CNT100 Offset,PR[24:Rotate_Offset] ;
4190:L P[2700]  R[157] mm/sec CNT100 Offset,PR[24:Rotate_Offset] ;
4191: !Pass212 ;
4192: LBL[1212:Pass212] ;
4193:L P[2701]  R[157] mm/sec FINE Offset,PR[78:Offst_apprch]  ;
4194: WAIT   0.20(sec) ;
4195:L P[2701]  R[157] mm/sec CNT100 TA    0.00sec,CALL RUN_LASER_START Offset,PR[25:Start_Offset] ;
4197:L P[2702]  R[157] mm/sec CNT100 Offset,PR[24:Rotate_Offset] ;
4198:L P[2703]  R[157] mm/sec CNT100 TA    0.00sec,CALL RUN_LASER_STOP Offset,PR[26:Stop_Offset] ;
4200:L P[2703]  R[157] mm/sec FINE Offset,PR[76:Offst_dprt] ;
4201:L P[2704]  R[157] mm/sec CNT100 Offset,PR[24:Rotate_Offset] ;
4202:L P[2705]  R[157] mm/sec CNT100 Offset,PR[24:Rotate_Offset] ;
4203:L P[2706]  R[157] mm/sec CNT100 Offset,PR[24:Rotate_Offset] ;
4204:L P[2707]  R[157] mm/sec CNT100 Offset,PR[24:Rotate_Offset] ;
4205:L P[2708]  R[157] mm/sec CNT100 Offset,PR[24:Rotate_Offset] ;
4206:L P[2709]  R[157] mm/sec CNT100 Offset,PR[24:Rotate_Offset] ;
4207: !Pass213 ;
4208: LBL[1213:Pass213] ;
4209:L P[2710]  R[157] mm/sec FINE Offset,PR[78:Offst_apprch]  ;
4210: WAIT   0.20(sec) ;
4211:L P[2710]  R[157] mm/sec CNT100 TA    0.00sec,CALL RUN_LASER_START Offset,PR[25:Start_Offset] ;
4213:L P[2711]  R[157] mm/sec CNT100 Offset,PR[24:Rotate_Offset] ;
4214:L P[2712]  R[157] mm/sec CNT100 Offset,PR[24:Rotate_Offset] ;
4215:L P[2713]  R[157] mm/sec CNT100 Offset,PR[24:Rotate_Offset] ;
4216:L P[2714]  R[157] mm/sec CNT100 TA    0.00sec,CALL RUN_LASER_STOP Offset,PR[26:Stop_Offset] ;
4218:L P[2714]  R[157] mm/sec FINE Offset,PR[76:Offst_dprt] ;
4219:L P[2715]  R[157] mm/sec CNT100 Offset,PR[24:Rotate_Offset] ;
4220:L P[2716]  R[157] mm/sec CNT100 Offset,PR[24:Rotate_Offset] ;
4221:L P[2717]  R[157] mm/sec CNT100 Offset,PR[24:Rotate_Offset] ;
4222:L P[2718]  R[157] mm/sec CNT100 Offset,PR[24:Rotate_Offset] ;
4223:L P[2719]  R[157] mm/sec CNT100 Offset,PR[24:Rotate_Offset] ;
4224:L P[2720]  R[157] mm/sec CNT100 Offset,PR[24:Rotate_Offset] ;
4225: !Pass214 ;
4226: LBL[1214:Pass214] ;
4227:L P[2721]  R[157] mm/sec FINE Offset,PR[78:Offst_apprch]  ;
4228: WAIT   0.20(sec) ;
4229:L P[2721]  R[157] mm/sec CNT100 TA    0.00sec,CALL RUN_LASER_START Offset,PR[25:Start_Offset] ;
4231:L P[2722]  R[157] mm/sec CNT100 Offset,PR[24:Rotate_Offset] ;
4232:L P[2723]  R[157] mm/sec CNT100 Offset,PR[24:Rotate_Offset] ;
4233:L P[2724]  R[157] mm/sec CNT100 Offset,PR[24:Rotate_Offset] ;
4234:L P[2725]  R[157] mm/sec CNT100 TA    0.00sec,CALL RUN_LASER_STOP Offset,PR[26:Stop_Offset] ;
4236:L P[2725]  R[157] mm/sec FINE Offset,PR[76:Offst_dprt] ;
4237:L P[2726]  R[157] mm/sec CNT100 Offset,PR[24:Rotate_Offset] ;
4238:L P[2727]  R[157] mm/sec CNT100 Offset,PR[24:Rotate_Offset] ;
4239:L P[2728]  R[157] mm/sec CNT100 Offset,PR[24:Rotate_Offset] ;
4240:L P[2729]  R[157] mm/sec CNT100 Offset,PR[24:Rotate_Offset] ;
4241:L P[2730]  R[157] mm/sec CNT100 Offset,PR[24:Rotate_Offset] ;
4242:L P[2731]  R[157] mm/sec CNT100 Offset,PR[24:Rotate_Offset] ;
4243: !Pass215 ;
4244: LBL[1215:Pass215] ;
4245:L P[2732]  R[157] mm/sec FINE Offset,PR[78:Offst_apprch]  ;
4246: WAIT   0.20(sec) ;
4247:L P[2732]  R[157] mm/sec CNT100 TA    0.00sec,CALL RUN_LASER_START Offset,PR[25:Start_Offset] ;
4249:L P[2733]  R[157] mm/sec CNT100 Offset,PR[24:Rotate_Offset] ;
4250:L P[2734]  R[157] mm/sec CNT100 Offset,PR[24:Rotate_Offset] ;
4251:L P[2735]  R[157] mm/sec CNT100 Offset,PR[24:Rotate_Offset] ;
4252:L P[2736]  R[157] mm/sec CNT100 TA    0.00sec,CALL RUN_LASER_STOP Offset,PR[26:Stop_Offset] ;
4254:L P[2736]  R[157] mm/sec FINE Offset,PR[76:Offst_dprt] ;
4255:L P[2737]  R[157] mm/sec CNT100 Offset,PR[24:Rotate_Offset] ;
4256:L P[2738]  R[157] mm/sec CNT100 Offset,PR[24:Rotate_Offset] ;
4257:L P[2739]  R[157] mm/sec CNT100 Offset,PR[24:Rotate_Offset] ;
4258:L P[2740]  R[157] mm/sec CNT100 Offset,PR[24:Rotate_Offset] ;
4259:L P[2741]  R[157] mm/sec CNT100 Offset,PR[24:Rotate_Offset] ;
4260:L P[2742]  R[157] mm/sec CNT100 Offset,PR[24:Rotate_Offset] ;
4261: !Pass216 ;
4262: LBL[1216:Pass216] ;
4263:L P[2743]  R[157] mm/sec FINE Offset,PR[78:Offst_apprch]  ;
4264: WAIT   0.20(sec) ;
4265:L P[2743]  R[157] mm/sec CNT100 TA    0.00sec,CALL RUN_LASER_START Offset,PR[25:Start_Offset] ;
4267:L P[2744]  R[157] mm/sec CNT100 Offset,PR[24:Rotate_Offset] ;
4268:L P[2745]  R[157] mm/sec CNT100 Offset,PR[24:Rotate_Offset] ;
4269:L P[2746]  R[157] mm/sec CNT100 Offset,PR[24:Rotate_Offset] ;
4270:L P[2747]  R[157] mm/sec CNT100 TA    0.00sec,CALL RUN_LASER_STOP Offset,PR[26:Stop_Offset] ;
4272:L P[2747]  R[157] mm/sec FINE Offset,PR[76:Offst_dprt] ;
4273:L P[2748]  R[157] mm/sec CNT100 Offset,PR[24:Rotate_Offset] ;
4274:L P[2749]  R[157] mm/sec CNT100 Offset,PR[24:Rotate_Offset] ;
4275:L P[2750]  R[157] mm/sec CNT100 Offset,PR[24:Rotate_Offset] ;
4276:L P[2751]  R[157] mm/sec CNT100 Offset,PR[24:Rotate_Offset] ;
4277:L P[2752]  R[157] mm/sec CNT100 Offset,PR[24:Rotate_Offset] ;
4278:L P[2753]  R[157] mm/sec CNT100 Offset,PR[24:Rotate_Offset] ;
4279: !Pass217 ;
4280: LBL[1217:Pass217] ;
4281:L P[2754]  R[157] mm/sec FINE Offset,PR[78:Offst_apprch]  ;
4282: WAIT   0.20(sec) ;
4283:L P[2754]  R[157] mm/sec CNT100 TA    0.00sec,CALL RUN_LASER_START Offset,PR[25:Start_Offset] ;
4285:L P[2755]  R[157] mm/sec CNT100 Offset,PR[24:Rotate_Offset] ;
4286:L P[2756]  R[157] mm/sec CNT100 Offset,PR[24:Rotate_Offset] ;
4287:L P[2757]  R[157] mm/sec CNT100 Offset,PR[24:Rotate_Offset] ;
4288:L P[2758]  R[157] mm/sec CNT100 Offset,PR[24:Rotate_Offset] ;
4289:L P[2759]  R[157] mm/sec CNT100 Offset,PR[24:Rotate_Offset] ;
4290:L P[2760]  R[157] mm/sec CNT100 TA    0.00sec,CALL RUN_LASER_STOP Offset,PR[26:Stop_Offset] ;
4292:L P[2760]  R[157] mm/sec FINE Offset,PR[76:Offst_dprt] ;
4293:L P[2761]  R[157] mm/sec CNT100 Offset,PR[24:Rotate_Offset] ;
4294:L P[2762]  R[157] mm/sec CNT100 Offset,PR[24:Rotate_Offset] ;
4295:L P[2763]  R[157] mm/sec CNT100 Offset,PR[24:Rotate_Offset] ;
4296:L P[2764]  R[157] mm/sec CNT100 Offset,PR[24:Rotate_Offset] ;
4297:L P[2765]  R[157] mm/sec CNT100 Offset,PR[24:Rotate_Offset] ;
4298:L P[2766]  R[157] mm/sec CNT100 Offset,PR[24:Rotate_Offset] ;
4299: !Pass218 ;
4300: LBL[1218:Pass218] ;
4301:L P[2767]  R[157] mm/sec FINE Offset,PR[78:Offst_apprch]  ;
4302: WAIT   0.20(sec) ;
4303:L P[2767]  R[157] mm/sec CNT100 TA    0.00sec,CALL RUN_LASER_START Offset,PR[25:Start_Offset] ;
4305:L P[2768]  R[157] mm/sec CNT100 Offset,PR[24:Rotate_Offset] ;
4306:L P[2769]  R[157] mm/sec CNT100 Offset,PR[24:Rotate_Offset] ;
4307:L P[2770]  R[157] mm/sec CNT100 Offset,PR[24:Rotate_Offset] ;
4308:L P[2771]  R[157] mm/sec CNT100 Offset,PR[24:Rotate_Offset] ;
4309:L P[2772]  R[157] mm/sec CNT100 TA    0.00sec,CALL RUN_LASER_STOP Offset,PR[26:Stop_Offset] ;
4311:L P[2772]  R[157] mm/sec FINE Offset,PR[76:Offst_dprt] ;
4312:L P[2773]  R[157] mm/sec CNT100 Offset,PR[24:Rotate_Offset] ;
4313:L P[2774]  R[157] mm/sec CNT100 Offset,PR[24:Rotate_Offset] ;
4314:L P[2775]  R[157] mm/sec CNT100 Offset,PR[24:Rotate_Offset] ;
4315:L P[2776]  R[157] mm/sec CNT100 Offset,PR[24:Rotate_Offset] ;
4316:L P[2777]  R[157] mm/sec CNT100 Offset,PR[24:Rotate_Offset] ;
4317:L P[2778]  R[157] mm/sec CNT100 Offset,PR[24:Rotate_Offset] ;
4318: !Pass219 ;
4319: LBL[1219:Pass219] ;
4320:L P[2779]  R[157] mm/sec FINE Offset,PR[78:Offst_apprch]  ;
4321: WAIT   0.20(sec) ;
4322:L P[2779]  R[157] mm/sec CNT100 TA    0.00sec,CALL RUN_LASER_START Offset,PR[25:Start_Offset] ;
4324:L P[2780]  R[157] mm/sec CNT100 Offset,PR[24:Rotate_Offset] ;
4325:L P[2781]  R[157] mm/sec CNT100 TA    0.00sec,CALL RUN_LASER_STOP Offset,PR[26:Stop_Offset] ;
4327:L P[2781]  R[157] mm/sec FINE Offset,PR[76:Offst_dprt] ;
4328:L P[2782]  R[157] mm/sec CNT100 Offset,PR[24:Rotate_Offset] ;
4329:L P[2783]  R[157] mm/sec CNT100 Offset,PR[24:Rotate_Offset] ;
4330:L P[2784]  R[157] mm/sec CNT100 Offset,PR[24:Rotate_Offset] ;
4331:L P[2785]  R[157] mm/sec CNT100 Offset,PR[24:Rotate_Offset] ;
4332:L P[2786]  R[157] mm/sec CNT100 Offset,PR[24:Rotate_Offset] ;
4333:L P[2787]  R[157] mm/sec CNT100 Offset,PR[24:Rotate_Offset] ;
4334: !Pass220 ;
4335: LBL[1220:Pass220] ;
4336:L P[2788]  R[157] mm/sec FINE Offset,PR[78:Offst_apprch]  ;
4337: WAIT   0.20(sec) ;
4338:L P[2788]  R[157] mm/sec CNT100 TA    0.00sec,CALL RUN_LASER_START Offset,PR[25:Start_Offset] ;
4340:L P[2789]  R[157] mm/sec CNT100 Offset,PR[24:Rotate_Offset] ;
4341:L P[2790]  R[157] mm/sec CNT100 TA    0.00sec,CALL RUN_LASER_STOP Offset,PR[26:Stop_Offset] ;
4343:L P[2790]  R[157] mm/sec FINE Offset,PR[76:Offst_dprt] ;
4344:L P[2791]  R[157] mm/sec CNT100 Offset,PR[24:Rotate_Offset] ;
4345:L P[2792]  R[157] mm/sec CNT100 Offset,PR[24:Rotate_Offset] ;
4346:L P[2793]  R[157] mm/sec CNT100 Offset,PR[24:Rotate_Offset] ;
4347:L P[2794]  R[157] mm/sec CNT100 Offset,PR[24:Rotate_Offset] ;
4348:L P[2795]  R[157] mm/sec CNT100 Offset,PR[24:Rotate_Offset] ;
4349:L P[2796]  R[157] mm/sec CNT100 Offset,PR[24:Rotate_Offset] ;
4350: !Pass221 ;
4351: LBL[1221:Pass221] ;
4352:L P[2797]  R[157] mm/sec FINE Offset,PR[78:Offst_apprch]  ;
4353: WAIT   0.20(sec) ;
4354:L P[2797]  R[157] mm/sec CNT100 TA    0.00sec,CALL RUN_LASER_START Offset,PR[25:Start_Offset] ;
4356:L P[2798]  R[157] mm/sec CNT100 Offset,PR[24:Rotate_Offset] ;
4357:L P[2799]  R[157] mm/sec CNT100 Offset,PR[24:Rotate_Offset] ;
4358:L P[2800]  R[157] mm/sec CNT100 Offset,PR[24:Rotate_Offset] ;
4359:L P[2801]  R[157] mm/sec CNT100 Offset,PR[24:Rotate_Offset] ;
4360:L P[2802]  R[157] mm/sec CNT100 Offset,PR[24:Rotate_Offset] ;
4361:L P[2803]  R[157] mm/sec CNT100 Offset,PR[24:Rotate_Offset] ;
4362:L P[2804]  R[157] mm/sec CNT100 TA    0.00sec,CALL RUN_LASER_STOP Offset,PR[26:Stop_Offset] ;
4364:L P[2804]  R[157] mm/sec FINE Offset,PR[76:Offst_dprt] ;
4365:L P[2805]  R[157] mm/sec CNT100 Offset,PR[24:Rotate_Offset] ;
4366:L P[2806]  R[157] mm/sec CNT100 Offset,PR[24:Rotate_Offset] ;
4367:L P[2807]  R[157] mm/sec CNT100 Offset,PR[24:Rotate_Offset] ;
4368:L P[2808]  R[157] mm/sec CNT100 Offset,PR[24:Rotate_Offset] ;
4369:L P[2809]  R[157] mm/sec CNT100 Offset,PR[24:Rotate_Offset] ;
4370:L P[2810]  R[157] mm/sec CNT100 Offset,PR[24:Rotate_Offset] ;
4371: !Pass222 ;
4372: LBL[1222:Pass222] ;
4373:L P[2811]  R[157] mm/sec FINE Offset,PR[78:Offst_apprch]  ;
4374: WAIT   0.20(sec) ;
4375:L P[2811]  R[157] mm/sec CNT100 TA    0.00sec,CALL RUN_LASER_START Offset,PR[25:Start_Offset] ;
4377:L P[2812]  R[157] mm/sec CNT100 Offset,PR[24:Rotate_Offset] ;
4378:L P[2813]  R[157] mm/sec CNT100 Offset,PR[24:Rotate_Offset] ;
4379:L P[2814]  R[157] mm/sec CNT100 Offset,PR[24:Rotate_Offset] ;
4380:L P[2815]  R[157] mm/sec CNT100 Offset,PR[24:Rotate_Offset] ;
4381:L P[2816]  R[157] mm/sec CNT100 Offset,PR[24:Rotate_Offset] ;
4382:L P[2817]  R[157] mm/sec CNT100 TA    0.00sec,CALL RUN_LASER_STOP Offset,PR[26:Stop_Offset] ;
4384:L P[2817]  R[157] mm/sec FINE Offset,PR[76:Offst_dprt] ;
4385:L P[2818]  R[157] mm/sec CNT100 Offset,PR[24:Rotate_Offset] ;
4386:L P[2819]  R[157] mm/sec CNT100 Offset,PR[24:Rotate_Offset] ;
4387:L P[2820]  R[157] mm/sec CNT100 Offset,PR[24:Rotate_Offset] ;
4388:L P[2821]  R[157] mm/sec CNT100 Offset,PR[24:Rotate_Offset] ;
4389:L P[2822]  R[157] mm/sec CNT100 Offset,PR[24:Rotate_Offset] ;
4390:L P[2823]  R[157] mm/sec CNT100 Offset,PR[24:Rotate_Offset] ;
4391: !Pass223 ;
4392: LBL[1223:Pass223] ;
4393:L P[2824]  R[157] mm/sec FINE Offset,PR[78:Offst_apprch]  ;
4394: WAIT   0.20(sec) ;
4395:L P[2824]  R[157] mm/sec CNT100 TA    0.00sec,CALL RUN_LASER_START Offset,PR[25:Start_Offset] ;
4397:L P[2825]  R[157] mm/sec CNT100 Offset,PR[24:Rotate_Offset] ;
4398:L P[2826]  R[157] mm/sec CNT100 Offset,PR[24:Rotate_Offset] ;
4399:L P[2827]  R[157] mm/sec CNT100 Offset,PR[24:Rotate_Offset] ;
4400:L P[2828]  R[157] mm/sec CNT100 Offset,PR[24:Rotate_Offset] ;
4401:L P[2829]  R[157] mm/sec CNT100 TA    0.00sec,CALL RUN_LASER_STOP Offset,PR[26:Stop_Offset] ;
4403:L P[2829]  R[157] mm/sec FINE Offset,PR[76:Offst_dprt] ;
4404:L P[2830]  R[157] mm/sec CNT100 Offset,PR[24:Rotate_Offset] ;
4405:L P[2831]  R[157] mm/sec CNT100 Offset,PR[24:Rotate_Offset] ;
4406:L P[2832]  R[157] mm/sec CNT100 Offset,PR[24:Rotate_Offset] ;
4407:L P[2833]  R[157] mm/sec CNT100 Offset,PR[24:Rotate_Offset] ;
4408:L P[2834]  R[157] mm/sec CNT100 Offset,PR[24:Rotate_Offset] ;
4409:L P[2835]  R[157] mm/sec CNT100 Offset,PR[24:Rotate_Offset] ;
4410: !Pass224 ;
4411: LBL[1224:Pass224] ;
4412:L P[2836]  R[157] mm/sec FINE Offset,PR[78:Offst_apprch]  ;
4413: WAIT   0.20(sec) ;
4414:L P[2836]  R[157] mm/sec CNT100 TA    0.00sec,CALL RUN_LASER_START Offset,PR[25:Start_Offset] ;
4416:L P[2837]  R[157] mm/sec CNT100 Offset,PR[24:Rotate_Offset] ;
4417:L P[2838]  R[157] mm/sec CNT100 Offset,PR[24:Rotate_Offset] ;
4418:L P[2839]  R[157] mm/sec CNT100 Offset,PR[24:Rotate_Offset] ;
4419:L P[2840]  R[157] mm/sec CNT100 Offset,PR[24:Rotate_Offset] ;
4420:L P[2841]  R[157] mm/sec CNT100 TA    0.00sec,CALL RUN_LASER_STOP Offset,PR[26:Stop_Offset] ;
4422:L P[2841]  R[157] mm/sec FINE Offset,PR[76:Offst_dprt] ;
4423:L P[2842]  R[157] mm/sec CNT100 Offset,PR[24:Rotate_Offset] ;
4424:L P[2843]  R[157] mm/sec CNT100 Offset,PR[24:Rotate_Offset] ;
4425:L P[2844]  R[157] mm/sec CNT100 Offset,PR[24:Rotate_Offset] ;
4426:L P[2845]  R[157] mm/sec CNT100 Offset,PR[24:Rotate_Offset] ;
4427:L P[2846]  R[157] mm/sec CNT100 Offset,PR[24:Rotate_Offset] ;
4428:L P[2847]  R[157] mm/sec CNT100 Offset,PR[24:Rotate_Offset] ;
4429: !Pass225 ;
4430: LBL[1225:Pass225] ;
4431:L P[2848]  R[157] mm/sec FINE Offset,PR[78:Offst_apprch]  ;
4432: WAIT   0.20(sec) ;
4433:L P[2848]  R[157] mm/sec CNT100 TA    0.00sec,CALL RUN_LASER_START Offset,PR[25:Start_Offset] ;
4435:L P[2849]  R[157] mm/sec CNT100 Offset,PR[24:Rotate_Offset] ;
4436:L P[2850]  R[157] mm/sec CNT100 Offset,PR[24:Rotate_Offset] ;
4437:L P[2851]  R[157] mm/sec CNT100 Offset,PR[24:Rotate_Offset] ;
4438:L P[2852]  R[157] mm/sec CNT100 Offset,PR[24:Rotate_Offset] ;
4439:L P[2853]  R[157] mm/sec CNT100 TA    0.00sec,CALL RUN_LASER_STOP Offset,PR[26:Stop_Offset] ;
4441:L P[2853]  R[157] mm/sec FINE Offset,PR[76:Offst_dprt] ;
4442:L P[2854]  R[157] mm/sec CNT100 Offset,PR[24:Rotate_Offset] ;
4443:L P[2855]  R[157] mm/sec CNT100 Offset,PR[24:Rotate_Offset] ;
4444:L P[2856]  R[157] mm/sec CNT100 Offset,PR[24:Rotate_Offset] ;
4445:L P[2857]  R[157] mm/sec CNT100 Offset,PR[24:Rotate_Offset] ;
4446:L P[2858]  R[157] mm/sec CNT100 Offset,PR[24:Rotate_Offset] ;
4447:L P[2859]  R[157] mm/sec CNT100 Offset,PR[24:Rotate_Offset] ;
4448: !Pass226 ;
4449: LBL[1226:Pass226] ;
4450:L P[2860]  R[157] mm/sec FINE Offset,PR[78:Offst_apprch]  ;
4451: WAIT   0.20(sec) ;
4452:L P[2860]  R[157] mm/sec CNT100 TA    0.00sec,CALL RUN_LASER_START Offset,PR[25:Start_Offset] ;
4454:L P[2861]  R[157] mm/sec CNT100 Offset,PR[24:Rotate_Offset] ;
4455:L P[2862]  R[157] mm/sec CNT100 Offset,PR[24:Rotate_Offset] ;
4456:L P[2863]  R[157] mm/sec CNT100 Offset,PR[24:Rotate_Offset] ;
4457:L P[2864]  R[157] mm/sec CNT100 Offset,PR[24:Rotate_Offset] ;
4458:L P[2865]  R[157] mm/sec CNT100 TA    0.00sec,CALL RUN_LASER_STOP Offset,PR[26:Stop_Offset] ;
4460:L P[2865]  R[157] mm/sec FINE Offset,PR[76:Offst_dprt] ;
4461:L P[2866]  R[157] mm/sec CNT100 Offset,PR[24:Rotate_Offset] ;
4462:L P[2867]  R[157] mm/sec CNT100 Offset,PR[24:Rotate_Offset] ;
4463:L P[2868]  R[157] mm/sec CNT100 Offset,PR[24:Rotate_Offset] ;
4464:L P[2869]  R[157] mm/sec CNT100 Offset,PR[24:Rotate_Offset] ;
4465:L P[2870]  R[157] mm/sec CNT100 Offset,PR[24:Rotate_Offset] ;
4466:L P[2871]  R[157] mm/sec CNT100 Offset,PR[24:Rotate_Offset] ;
4467: !Pass227 ;
4468: LBL[1227:Pass227] ;
4469:L P[2872]  R[157] mm/sec FINE Offset,PR[78:Offst_apprch]  ;
4470: WAIT   0.20(sec) ;
4471:L P[2872]  R[157] mm/sec CNT100 TA    0.00sec,CALL RUN_LASER_START Offset,PR[25:Start_Offset] ;
4473:L P[2873]  R[157] mm/sec CNT100 Offset,PR[24:Rotate_Offset] ;
4474:L P[2874]  R[157] mm/sec CNT100 TA    0.00sec,CALL RUN_LASER_STOP Offset,PR[26:Stop_Offset] ;
4476:L P[2874]  R[157] mm/sec FINE Offset,PR[76:Offst_dprt] ;
4477:L P[2875]  R[157] mm/sec CNT100 Offset,PR[24:Rotate_Offset] ;
4478:L P[2876]  R[157] mm/sec CNT100 Offset,PR[24:Rotate_Offset] ;
4479:L P[2877]  R[157] mm/sec CNT100 Offset,PR[24:Rotate_Offset] ;
4480:L P[2878]  R[157] mm/sec CNT100 Offset,PR[24:Rotate_Offset] ;
4481:L P[2879]  R[157] mm/sec CNT100 Offset,PR[24:Rotate_Offset] ;
4482:L P[2880]  R[157] mm/sec CNT100 Offset,PR[24:Rotate_Offset] ;
4483: !Pass228 ;
4484: LBL[1228:Pass228] ;
4485:L P[2881]  R[157] mm/sec FINE Offset,PR[78:Offst_apprch]  ;
4486: WAIT   0.20(sec) ;
4487:L P[2881]  R[157] mm/sec CNT100 TA    0.00sec,CALL RUN_LASER_START Offset,PR[25:Start_Offset] ;
4489:L P[2882]  R[157] mm/sec CNT100 Offset,PR[24:Rotate_Offset] ;
4490:L P[2883]  R[157] mm/sec CNT100 Offset,PR[24:Rotate_Offset] ;
4491:L P[2884]  R[157] mm/sec CNT100 TA    0.00sec,CALL RUN_LASER_STOP Offset,PR[26:Stop_Offset] ;
4493:L P[2884]  R[157] mm/sec FINE Offset,PR[76:Offst_dprt] ;
4494:L P[2885]  R[157] mm/sec CNT100 Offset,PR[24:Rotate_Offset] ;
4495:L P[2886]  R[157] mm/sec CNT100 Offset,PR[24:Rotate_Offset] ;
4496:L P[2887]  R[157] mm/sec CNT100 Offset,PR[24:Rotate_Offset] ;
4497:L P[2888]  R[157] mm/sec CNT100 Offset,PR[24:Rotate_Offset] ;
4498:L P[2889]  R[157] mm/sec CNT100 Offset,PR[24:Rotate_Offset] ;
4499:L P[2890]  R[157] mm/sec CNT100 Offset,PR[24:Rotate_Offset] ;
4500: !Pass229 ;
4501: LBL[1229:Pass229] ;
4502:L P[2891]  R[157] mm/sec FINE Offset,PR[78:Offst_apprch]  ;
4503: WAIT   0.20(sec) ;
4504:L P[2891]  R[157] mm/sec CNT100 TA    0.00sec,CALL RUN_LASER_START Offset,PR[25:Start_Offset] ;
4506:L P[2892]  R[157] mm/sec CNT100 Offset,PR[24:Rotate_Offset] ;
4507:L P[2893]  R[157] mm/sec CNT100 Offset,PR[24:Rotate_Offset] ;
4508:L P[2894]  R[157] mm/sec CNT100 Offset,PR[24:Rotate_Offset] ;
4509:L P[2895]  R[157] mm/sec CNT100 Offset,PR[24:Rotate_Offset] ;
4510:L P[2896]  R[157] mm/sec CNT100 TA    0.00sec,CALL RUN_LASER_STOP Offset,PR[26:Stop_Offset] ;
4512:L P[2896]  R[157] mm/sec FINE Offset,PR[76:Offst_dprt] ;
4513:L P[2897]  R[157] mm/sec CNT100 Offset,PR[24:Rotate_Offset] ;
4514:L P[2898]  R[157] mm/sec CNT100 Offset,PR[24:Rotate_Offset] ;
4515:L P[2899]  R[157] mm/sec CNT100 Offset,PR[24:Rotate_Offset] ;
4516:L P[2900]  R[157] mm/sec CNT100 Offset,PR[24:Rotate_Offset] ;
4517:L P[2901]  R[157] mm/sec CNT100 Offset,PR[24:Rotate_Offset] ;
4518:L P[2902]  R[157] mm/sec CNT100 Offset,PR[24:Rotate_Offset] ;
4519: !Pass230 ;
4520: LBL[1230:Pass230] ;
4521:L P[2903]  R[157] mm/sec FINE Offset,PR[78:Offst_apprch]  ;
4522: WAIT   0.20(sec) ;
4523:L P[2903]  R[157] mm/sec CNT100 TA    0.00sec,CALL RUN_LASER_START Offset,PR[25:Start_Offset] ;
4525:L P[2904]  R[157] mm/sec CNT100 Offset,PR[24:Rotate_Offset] ;
4526:L P[2905]  R[157] mm/sec CNT100 Offset,PR[24:Rotate_Offset] ;
4527:L P[2906]  R[157] mm/sec CNT100 Offset,PR[24:Rotate_Offset] ;
4528:L P[2907]  R[157] mm/sec CNT100 Offset,PR[24:Rotate_Offset] ;
4529:L P[2908]  R[157] mm/sec CNT100 TA    0.00sec,CALL RUN_LASER_STOP Offset,PR[26:Stop_Offset] ;
4531:L P[2908]  R[157] mm/sec FINE Offset,PR[76:Offst_dprt] ;
4532:L P[2909]  R[157] mm/sec CNT100 Offset,PR[24:Rotate_Offset] ;
4533:L P[2910]  R[157] mm/sec CNT100 Offset,PR[24:Rotate_Offset] ;
4534:L P[2911]  R[157] mm/sec CNT100 Offset,PR[24:Rotate_Offset] ;
4535:L P[2912]  R[157] mm/sec CNT100 Offset,PR[24:Rotate_Offset] ;
4536:L P[2913]  R[157] mm/sec CNT100 Offset,PR[24:Rotate_Offset] ;
4537:L P[2914]  R[157] mm/sec CNT100 Offset,PR[24:Rotate_Offset] ;
4538: !Pass231 ;
4539: LBL[1231:Pass231] ;
4540:L P[2915]  R[157] mm/sec FINE Offset,PR[78:Offst_apprch]  ;
4541: WAIT   0.20(sec) ;
4542:L P[2915]  R[157] mm/sec CNT100 TA    0.00sec,CALL RUN_LASER_START Offset,PR[25:Start_Offset] ;
4544:L P[2916]  R[157] mm/sec CNT100 Offset,PR[24:Rotate_Offset] ;
4545:L P[2917]  R[157] mm/sec CNT100 Offset,PR[24:Rotate_Offset] ;
4546:L P[2918]  R[157] mm/sec CNT100 Offset,PR[24:Rotate_Offset] ;
4547:L P[2919]  R[157] mm/sec CNT100 Offset,PR[24:Rotate_Offset] ;
4548:L P[2920]  R[157] mm/sec CNT100 TA    0.00sec,CALL RUN_LASER_STOP Offset,PR[26:Stop_Offset] ;
4550:L P[2920]  R[157] mm/sec FINE Offset,PR[76:Offst_dprt] ;
4551:L P[2921]  R[157] mm/sec CNT100 Offset,PR[24:Rotate_Offset] ;
4552:L P[2922]  R[157] mm/sec CNT100 Offset,PR[24:Rotate_Offset] ;
4553:L P[2923]  R[157] mm/sec CNT100 Offset,PR[24:Rotate_Offset] ;
4554:L P[2924]  R[157] mm/sec CNT100 Offset,PR[24:Rotate_Offset] ;
4555:L P[2925]  R[157] mm/sec CNT100 Offset,PR[24:Rotate_Offset] ;
4556:L P[2926]  R[157] mm/sec CNT100 Offset,PR[24:Rotate_Offset] ;
4557: !Pass232 ;
4558: LBL[1232:Pass232] ;
4559:L P[2927]  R[157] mm/sec FINE Offset,PR[78:Offst_apprch]  ;
4560: WAIT   0.20(sec) ;
4561:L P[2927]  R[157] mm/sec CNT100 TA    0.00sec,CALL RUN_LASER_START Offset,PR[25:Start_Offset] ;
4563:L P[2928]  R[157] mm/sec CNT100 Offset,PR[24:Rotate_Offset] ;
4564:L P[2929]  R[157] mm/sec CNT100 Offset,PR[24:Rotate_Offset] ;
4565:L P[2930]  R[157] mm/sec CNT100 Offset,PR[24:Rotate_Offset] ;
4566:L P[2931]  R[157] mm/sec CNT100 Offset,PR[24:Rotate_Offset] ;
4567:L P[2932]  R[157] mm/sec CNT100 TA    0.00sec,CALL RUN_LASER_STOP Offset,PR[26:Stop_Offset] ;
4569:L P[2932]  R[157] mm/sec FINE Offset,PR[76:Offst_dprt] ;
4570:L P[2933]  R[157] mm/sec CNT100 Offset,PR[24:Rotate_Offset] ;
4571:L P[2934]  R[157] mm/sec CNT100 Offset,PR[24:Rotate_Offset] ;
4572:L P[2935]  R[157] mm/sec CNT100 Offset,PR[24:Rotate_Offset] ;
4573:L P[2936]  R[157] mm/sec CNT100 Offset,PR[24:Rotate_Offset] ;
4574:L P[2937]  R[157] mm/sec CNT100 Offset,PR[24:Rotate_Offset] ;
4575:L P[2938]  R[157] mm/sec CNT100 Offset,PR[24:Rotate_Offset] ;
4576: !Pass233 ;
4577: LBL[1233:Pass233] ;
4578:L P[2939]  R[157] mm/sec FINE Offset,PR[78:Offst_apprch]  ;
4579: WAIT   0.20(sec) ;
4580:L P[2939]  R[157] mm/sec CNT100 TA    0.00sec,CALL RUN_LASER_START Offset,PR[25:Start_Offset] ;
4582:L P[2940]  R[157] mm/sec CNT100 Offset,PR[24:Rotate_Offset] ;
4583:L P[2941]  R[157] mm/sec CNT100 Offset,PR[24:Rotate_Offset] ;
4584:L P[2942]  R[157] mm/sec CNT100 Offset,PR[24:Rotate_Offset] ;
4585:L P[2943]  R[157] mm/sec CNT100 Offset,PR[24:Rotate_Offset] ;
4586:L P[2944]  R[157] mm/sec CNT100 Offset,PR[24:Rotate_Offset] ;
4587:L P[2945]  R[157] mm/sec CNT100 Offset,PR[24:Rotate_Offset] ;
4588:L P[2946]  R[157] mm/sec CNT100 TA    0.00sec,CALL RUN_LASER_STOP Offset,PR[26:Stop_Offset] ;
4590:L P[2946]  R[157] mm/sec FINE Offset,PR[76:Offst_dprt] ;
4591:L P[2947]  R[157] mm/sec CNT100 Offset,PR[24:Rotate_Offset] ;
4592:L P[2948]  R[157] mm/sec CNT100 Offset,PR[24:Rotate_Offset] ;
4593:L P[2949]  R[157] mm/sec CNT100 Offset,PR[24:Rotate_Offset] ;
4594:L P[2950]  R[157] mm/sec CNT100 Offset,PR[24:Rotate_Offset] ;
4595:L P[2951]  R[157] mm/sec CNT100 Offset,PR[24:Rotate_Offset] ;
4596:L P[2952]  R[157] mm/sec CNT100 Offset,PR[24:Rotate_Offset] ;
4597: !Pass234 ;
4598: LBL[1234:Pass234] ;
4599:L P[2953]  R[157] mm/sec FINE Offset,PR[78:Offst_apprch]  ;
4600: WAIT   0.20(sec) ;
4601:L P[2953]  R[157] mm/sec CNT100 TA    0.00sec,CALL RUN_LASER_START Offset,PR[25:Start_Offset] ;
4603:L P[2954]  R[157] mm/sec CNT100 Offset,PR[24:Rotate_Offset] ;
4604:L P[2955]  R[157] mm/sec CNT100 Offset,PR[24:Rotate_Offset] ;
4605:L P[2956]  R[157] mm/sec CNT100 Offset,PR[24:Rotate_Offset] ;
4606:L P[2957]  R[157] mm/sec CNT100 Offset,PR[24:Rotate_Offset] ;
4607:L P[2958]  R[157] mm/sec CNT100 Offset,PR[24:Rotate_Offset] ;
4608:L P[2959]  R[157] mm/sec CNT100 Offset,PR[24:Rotate_Offset] ;
4609:L P[2960]  R[157] mm/sec CNT100 TA    0.00sec,CALL RUN_LASER_STOP Offset,PR[26:Stop_Offset] ;
4611:L P[2960]  R[157] mm/sec FINE Offset,PR[76:Offst_dprt] ;
4612:L P[2961]  R[157] mm/sec CNT100 Offset,PR[24:Rotate_Offset] ;
4613:L P[2962]  R[157] mm/sec CNT100 Offset,PR[24:Rotate_Offset] ;
4614:L P[2963]  R[157] mm/sec CNT100 Offset,PR[24:Rotate_Offset] ;
4615:L P[2964]  R[157] mm/sec CNT100 Offset,PR[24:Rotate_Offset] ;
4616:L P[2965]  R[157] mm/sec CNT100 Offset,PR[24:Rotate_Offset] ;
4617:L P[2966]  R[157] mm/sec CNT100 Offset,PR[24:Rotate_Offset] ;
4618: !Pass235 ;
4619: LBL[1235:Pass235] ;
4620:L P[2967]  R[157] mm/sec FINE Offset,PR[78:Offst_apprch]  ;
4621: WAIT   0.20(sec) ;
4622:L P[2967]  R[157] mm/sec CNT100 TA    0.00sec,CALL RUN_LASER_START Offset,PR[25:Start_Offset] ;
4624:L P[2968]  R[157] mm/sec CNT100 Offset,PR[24:Rotate_Offset] ;
4625:L P[2969]  R[157] mm/sec CNT100 Offset,PR[24:Rotate_Offset] ;
4626:L P[2970]  R[157] mm/sec CNT100 TA    0.00sec,CALL RUN_LASER_STOP Offset,PR[26:Stop_Offset] ;
4628:L P[2970]  R[157] mm/sec FINE Offset,PR[76:Offst_dprt] ;
4629:L P[2971]  R[157] mm/sec CNT100 Offset,PR[24:Rotate_Offset] ;
4630:L P[2972]  R[157] mm/sec CNT100 Offset,PR[24:Rotate_Offset] ;
4631:L P[2973]  R[157] mm/sec CNT100 Offset,PR[24:Rotate_Offset] ;
4632:L P[2974]  R[157] mm/sec CNT100 Offset,PR[24:Rotate_Offset] ;
4633:L P[2975]  R[157] mm/sec CNT100 Offset,PR[24:Rotate_Offset] ;
4634:L P[2976]  R[157] mm/sec CNT100 Offset,PR[24:Rotate_Offset] ;
4635: !Pass236 ;
4636: LBL[1236:Pass236] ;
4637:L P[2977]  R[157] mm/sec FINE Offset,PR[78:Offst_apprch]  ;
4638: WAIT   0.20(sec) ;
4639:L P[2977]  R[157] mm/sec CNT100 TA    0.00sec,CALL RUN_LASER_START Offset,PR[25:Start_Offset] ;
4641:L P[2978]  R[157] mm/sec CNT100 Offset,PR[24:Rotate_Offset] ;
4642:L P[2979]  R[157] mm/sec CNT100 Offset,PR[24:Rotate_Offset] ;
4643:L P[2980]  R[157] mm/sec CNT100 Offset,PR[24:Rotate_Offset] ;
4644:L P[2981]  R[157] mm/sec CNT100 Offset,PR[24:Rotate_Offset] ;
4645:L P[2982]  R[157] mm/sec CNT100 Offset,PR[24:Rotate_Offset] ;
4646:L P[2983]  R[157] mm/sec CNT100 Offset,PR[24:Rotate_Offset] ;
4647:L P[2984]  R[157] mm/sec CNT100 Offset,PR[24:Rotate_Offset] ;
4648:L P[2985]  R[157] mm/sec CNT100 Offset,PR[24:Rotate_Offset] ;
4649:L P[2986]  R[157] mm/sec CNT100 Offset,PR[24:Rotate_Offset] ;
4650:L P[2987]  R[157] mm/sec CNT100 Offset,PR[24:Rotate_Offset] ;
4651:L P[2988]  R[157] mm/sec CNT100 Offset,PR[24:Rotate_Offset] ;
4652:L P[2989]  R[157] mm/sec CNT100 Offset,PR[24:Rotate_Offset] ;
4653:L P[2990]  R[157] mm/sec CNT100 Offset,PR[24:Rotate_Offset] ;
4654:L P[2991]  R[157] mm/sec CNT100 Offset,PR[24:Rotate_Offset] ;
4655:L P[2992]  R[157] mm/sec CNT100 Offset,PR[24:Rotate_Offset] ;
4656:L P[2993]  R[157] mm/sec CNT100 Offset,PR[24:Rotate_Offset] ;
4657:L P[2994]  R[157] mm/sec CNT100 Offset,PR[24:Rotate_Offset] ;
4658:L P[2995]  R[157] mm/sec CNT100 Offset,PR[24:Rotate_Offset] ;
4659:L P[2996]  R[157] mm/sec CNT100 Offset,PR[24:Rotate_Offset] ;
4660:L P[2997]  R[157] mm/sec CNT100 Offset,PR[24:Rotate_Offset] ;
4661:L P[2998]  R[157] mm/sec CNT100 Offset,PR[24:Rotate_Offset] ;
4662:L P[2999]  R[157] mm/sec CNT100 Offset,PR[24:Rotate_Offset] ;
4663:L P[3000]  R[157] mm/sec CNT100 Offset,PR[24:Rotate_Offset] ;
4664:L P[3001]  R[157] mm/sec CNT100 Offset,PR[24:Rotate_Offset] ;
4665:L P[3002]  R[157] mm/sec CNT100 Offset,PR[24:Rotate_Offset] ;
4666:L P[3003]  R[157] mm/sec CNT100 Offset,PR[24:Rotate_Offset] ;
4667:L P[3004]  R[157] mm/sec CNT100 Offset,PR[24:Rotate_Offset] ;
4668:L P[3005]  R[157] mm/sec CNT100 Offset,PR[24:Rotate_Offset] ;
4669:L P[3006]  R[157] mm/sec CNT100 Offset,PR[24:Rotate_Offset] ;
4670:L P[3007]  R[157] mm/sec CNT100 Offset,PR[24:Rotate_Offset] ;
4671:L P[3008]  R[157] mm/sec CNT100 Offset,PR[24:Rotate_Offset] ;
4672:L P[3009]  R[157] mm/sec CNT100 Offset,PR[24:Rotate_Offset] ;
4673:L P[3010]  R[157] mm/sec CNT100 Offset,PR[24:Rotate_Offset] ;
4674:L P[3011]  R[157] mm/sec CNT100 Offset,PR[24:Rotate_Offset] ;
4675:L P[3012]  R[157] mm/sec CNT100 Offset,PR[24:Rotate_Offset] ;
4676:L P[3013]  R[157] mm/sec CNT100 Offset,PR[24:Rotate_Offset] ;
4677:L P[3014]  R[157] mm/sec CNT100 Offset,PR[24:Rotate_Offset] ;
4678:L P[3015]  R[157] mm/sec CNT100 Offset,PR[24:Rotate_Offset] ;
4679:L P[3016]  R[157] mm/sec CNT100 Offset,PR[24:Rotate_Offset] ;
4680:L P[3017]  R[157] mm/sec CNT100 Offset,PR[24:Rotate_Offset] ;
4681:L P[3018]  R[157] mm/sec CNT100 Offset,PR[24:Rotate_Offset] ;
4682:L P[3019]  R[157] mm/sec CNT100 Offset,PR[24:Rotate_Offset] ;
4683:L P[3020]  R[157] mm/sec CNT100 Offset,PR[24:Rotate_Offset] ;
4684:L P[3021]  R[157] mm/sec CNT100 Offset,PR[24:Rotate_Offset] ;
4685:L P[3022]  R[157] mm/sec CNT100 Offset,PR[24:Rotate_Offset] ;
4686:L P[3023]  R[157] mm/sec CNT100 Offset,PR[24:Rotate_Offset] ;
4687:L P[3024]  R[157] mm/sec CNT100 Offset,PR[24:Rotate_Offset] ;
4688:L P[3025]  R[157] mm/sec CNT100 Offset,PR[24:Rotate_Offset] ;
4689:L P[3026]  R[157] mm/sec CNT100 Offset,PR[24:Rotate_Offset] ;
4690:L P[3027]  R[157] mm/sec CNT100 Offset,PR[24:Rotate_Offset] ;
4691:L P[3028]  R[157] mm/sec CNT100 TA    0.00sec,CALL RUN_LASER_STOP Offset,PR[26:Stop_Offset] ;
4693:L P[3028]  R[157] mm/sec FINE Offset,PR[76:Offst_dprt] ;
4694:L P[3029]  R[157] mm/sec CNT100 Offset,PR[24:Rotate_Offset] ;
4695:L P[3030]  R[157] mm/sec CNT100 Offset,PR[24:Rotate_Offset] ;
4696:L P[3031]  R[157] mm/sec CNT100 Offset,PR[24:Rotate_Offset] ;
4697:L P[3032]  R[157] mm/sec CNT100 Offset,PR[24:Rotate_Offset] ;
4698:L P[3033]  R[157] mm/sec CNT100 Offset,PR[24:Rotate_Offset] ;
4699:L P[3034]  R[157] mm/sec CNT100 Offset,PR[24:Rotate_Offset] ;
4700: !Pass237 ;
4701: LBL[1237:Pass237] ;
4702:L P[3035]  R[157] mm/sec FINE Offset,PR[78:Offst_apprch]  ;
4703: WAIT   0.20(sec) ;
4704:L P[3035]  R[157] mm/sec CNT100 TA    0.00sec,CALL RUN_LASER_START Offset,PR[25:Start_Offset] ;
4706:L P[3036]  R[157] mm/sec CNT100 Offset,PR[24:Rotate_Offset] ;
4707:L P[3037]  R[157] mm/sec CNT100 Offset,PR[24:Rotate_Offset] ;
4708:L P[3038]  R[157] mm/sec CNT100 Offset,PR[24:Rotate_Offset] ;
4709:L P[3039]  R[157] mm/sec CNT100 Offset,PR[24:Rotate_Offset] ;
4710:L P[3040]  R[157] mm/sec CNT100 Offset,PR[24:Rotate_Offset] ;
4711:L P[3041]  R[157] mm/sec CNT100 Offset,PR[24:Rotate_Offset] ;
4712:L P[3042]  R[157] mm/sec CNT100 Offset,PR[24:Rotate_Offset] ;
4713:L P[3043]  R[157] mm/sec CNT100 Offset,PR[24:Rotate_Offset] ;
4714:L P[3044]  R[157] mm/sec CNT100 Offset,PR[24:Rotate_Offset] ;
4715:L P[3045]  R[157] mm/sec CNT100 Offset,PR[24:Rotate_Offset] ;
4716:L P[3046]  R[157] mm/sec CNT100 Offset,PR[24:Rotate_Offset] ;
4717:L P[3047]  R[157] mm/sec CNT100 Offset,PR[24:Rotate_Offset] ;
4718:L P[3048]  R[157] mm/sec CNT100 Offset,PR[24:Rotate_Offset] ;
4719:L P[3049]  R[157] mm/sec CNT100 Offset,PR[24:Rotate_Offset] ;
4720:L P[3050]  R[157] mm/sec CNT100 Offset,PR[24:Rotate_Offset] ;
4721:L P[3051]  R[157] mm/sec CNT100 Offset,PR[24:Rotate_Offset] ;
4722:L P[3052]  R[157] mm/sec CNT100 Offset,PR[24:Rotate_Offset] ;
4723:L P[3053]  R[157] mm/sec CNT100 Offset,PR[24:Rotate_Offset] ;
4724:L P[3054]  R[157] mm/sec CNT100 Offset,PR[24:Rotate_Offset] ;
4725:L P[3055]  R[157] mm/sec CNT100 Offset,PR[24:Rotate_Offset] ;
4726:L P[3056]  R[157] mm/sec CNT100 Offset,PR[24:Rotate_Offset] ;
4727:L P[3057]  R[157] mm/sec CNT100 Offset,PR[24:Rotate_Offset] ;
4728:L P[3058]  R[157] mm/sec CNT100 Offset,PR[24:Rotate_Offset] ;
4729:L P[3059]  R[157] mm/sec CNT100 Offset,PR[24:Rotate_Offset] ;
4730:L P[3060]  R[157] mm/sec CNT100 Offset,PR[24:Rotate_Offset] ;
4731:L P[3061]  R[157] mm/sec CNT100 Offset,PR[24:Rotate_Offset] ;
4732:L P[3062]  R[157] mm/sec CNT100 Offset,PR[24:Rotate_Offset] ;
4733:L P[3063]  R[157] mm/sec CNT100 Offset,PR[24:Rotate_Offset] ;
4734:L P[3064]  R[157] mm/sec CNT100 Offset,PR[24:Rotate_Offset] ;
4735:L P[3065]  R[157] mm/sec CNT100 Offset,PR[24:Rotate_Offset] ;
4736:L P[3066]  R[157] mm/sec CNT100 Offset,PR[24:Rotate_Offset] ;
4737:L P[3067]  R[157] mm/sec CNT100 Offset,PR[24:Rotate_Offset] ;
4738:L P[3068]  R[157] mm/sec CNT100 Offset,PR[24:Rotate_Offset] ;
4739:L P[3069]  R[157] mm/sec CNT100 Offset,PR[24:Rotate_Offset] ;
4740:L P[3070]  R[157] mm/sec CNT100 Offset,PR[24:Rotate_Offset] ;
4741:L P[3071]  R[157] mm/sec CNT100 Offset,PR[24:Rotate_Offset] ;
4742:L P[3072]  R[157] mm/sec CNT100 Offset,PR[24:Rotate_Offset] ;
4743:L P[3073]  R[157] mm/sec CNT100 Offset,PR[24:Rotate_Offset] ;
4744:L P[3074]  R[157] mm/sec CNT100 Offset,PR[24:Rotate_Offset] ;
4745:L P[3075]  R[157] mm/sec CNT100 Offset,PR[24:Rotate_Offset] ;
4746:L P[3076]  R[157] mm/sec CNT100 Offset,PR[24:Rotate_Offset] ;
4747:L P[3077]  R[157] mm/sec CNT100 Offset,PR[24:Rotate_Offset] ;
4748:L P[3078]  R[157] mm/sec CNT100 Offset,PR[24:Rotate_Offset] ;
4749:L P[3079]  R[157] mm/sec CNT100 Offset,PR[24:Rotate_Offset] ;
4750:L P[3080]  R[157] mm/sec CNT100 Offset,PR[24:Rotate_Offset] ;
4751:L P[3081]  R[157] mm/sec CNT100 Offset,PR[24:Rotate_Offset] ;
4752:L P[3082]  R[157] mm/sec CNT100 Offset,PR[24:Rotate_Offset] ;
4753:L P[3083]  R[157] mm/sec CNT100 Offset,PR[24:Rotate_Offset] ;
4754:L P[3084]  R[157] mm/sec CNT100 Offset,PR[24:Rotate_Offset] ;
4755:L P[3085]  R[157] mm/sec CNT100 Offset,PR[24:Rotate_Offset] ;
4756:L P[3086]  R[157] mm/sec CNT100 TA    0.00sec,CALL RUN_LASER_STOP Offset,PR[26:Stop_Offset] ;
4758:L P[3086]  R[157] mm/sec FINE Offset,PR[76:Offst_dprt] ;
4759:L P[3087]  R[157] mm/sec CNT100 Offset,PR[24:Rotate_Offset] ;
4760:L P[3088]  R[157] mm/sec CNT100 Offset,PR[24:Rotate_Offset] ;
4761:L P[3089]  R[157] mm/sec CNT100 Offset,PR[24:Rotate_Offset] ;
4762:L P[3090]  R[157] mm/sec CNT100 Offset,PR[24:Rotate_Offset] ;
4763:L P[3091]  R[157] mm/sec CNT100 Offset,PR[24:Rotate_Offset] ;
4764:L P[3092]  R[157] mm/sec CNT100 Offset,PR[24:Rotate_Offset] ;
4765: !Pass238 ;
4766: LBL[1238:Pass238] ;
4767:L P[3093]  R[157] mm/sec FINE Offset,PR[78:Offst_apprch]  ;
4768: WAIT   0.20(sec) ;
4769:L P[3093]  R[157] mm/sec CNT100 TA    0.00sec,CALL RUN_LASER_START Offset,PR[25:Start_Offset] ;
4771:L P[3094]  R[157] mm/sec CNT100 Offset,PR[24:Rotate_Offset] ;
4772:L P[3095]  R[157] mm/sec CNT100 Offset,PR[24:Rotate_Offset] ;
4773:L P[3096]  R[157] mm/sec CNT100 Offset,PR[24:Rotate_Offset] ;
4774:L P[3097]  R[157] mm/sec CNT100 Offset,PR[24:Rotate_Offset] ;
4775:L P[3098]  R[157] mm/sec CNT100 Offset,PR[24:Rotate_Offset] ;
4776:L P[3099]  R[157] mm/sec CNT100 Offset,PR[24:Rotate_Offset] ;
4777:L P[3100]  R[157] mm/sec CNT100 Offset,PR[24:Rotate_Offset] ;
4778:L P[3101]  R[157] mm/sec CNT100 Offset,PR[24:Rotate_Offset] ;
4779:L P[3102]  R[157] mm/sec CNT100 Offset,PR[24:Rotate_Offset] ;
4780:L P[3103]  R[157] mm/sec CNT100 Offset,PR[24:Rotate_Offset] ;
4781:L P[3104]  R[157] mm/sec CNT100 Offset,PR[24:Rotate_Offset] ;
4782:L P[3105]  R[157] mm/sec CNT100 Offset,PR[24:Rotate_Offset] ;
4783:L P[3106]  R[157] mm/sec CNT100 Offset,PR[24:Rotate_Offset] ;
4784:L P[3107]  R[157] mm/sec CNT100 Offset,PR[24:Rotate_Offset] ;
4785:L P[3108]  R[157] mm/sec CNT100 Offset,PR[24:Rotate_Offset] ;
4786:L P[3109]  R[157] mm/sec CNT100 Offset,PR[24:Rotate_Offset] ;
4787:L P[3110]  R[157] mm/sec CNT100 Offset,PR[24:Rotate_Offset] ;
4788:L P[3111]  R[157] mm/sec CNT100 Offset,PR[24:Rotate_Offset] ;
4789:L P[3112]  R[157] mm/sec CNT100 Offset,PR[24:Rotate_Offset] ;
4790:L P[3113]  R[157] mm/sec CNT100 Offset,PR[24:Rotate_Offset] ;
4791:L P[3114]  R[157] mm/sec CNT100 Offset,PR[24:Rotate_Offset] ;
4792:L P[3115]  R[157] mm/sec CNT100 Offset,PR[24:Rotate_Offset] ;
4793:L P[3116]  R[157] mm/sec CNT100 Offset,PR[24:Rotate_Offset] ;
4794:L P[3117]  R[157] mm/sec CNT100 Offset,PR[24:Rotate_Offset] ;
4795:L P[3118]  R[157] mm/sec CNT100 Offset,PR[24:Rotate_Offset] ;
4796:L P[3119]  R[157] mm/sec CNT100 Offset,PR[24:Rotate_Offset] ;
4797:L P[3120]  R[157] mm/sec CNT100 Offset,PR[24:Rotate_Offset] ;
4798:L P[3121]  R[157] mm/sec CNT100 Offset,PR[24:Rotate_Offset] ;
4799:L P[3122]  R[157] mm/sec CNT100 Offset,PR[24:Rotate_Offset] ;
4800:L P[3123]  R[157] mm/sec CNT100 Offset,PR[24:Rotate_Offset] ;
4801:L P[3124]  R[157] mm/sec CNT100 Offset,PR[24:Rotate_Offset] ;
4802:L P[3125]  R[157] mm/sec CNT100 Offset,PR[24:Rotate_Offset] ;
4803:L P[3126]  R[157] mm/sec CNT100 Offset,PR[24:Rotate_Offset] ;
4804:L P[3127]  R[157] mm/sec CNT100 Offset,PR[24:Rotate_Offset] ;
4805:L P[3128]  R[157] mm/sec CNT100 Offset,PR[24:Rotate_Offset] ;
4806:L P[3129]  R[157] mm/sec CNT100 Offset,PR[24:Rotate_Offset] ;
4807:L P[3130]  R[157] mm/sec CNT100 Offset,PR[24:Rotate_Offset] ;
4808:L P[3131]  R[157] mm/sec CNT100 Offset,PR[24:Rotate_Offset] ;
4809:L P[3132]  R[157] mm/sec CNT100 Offset,PR[24:Rotate_Offset] ;
4810:L P[3133]  R[157] mm/sec CNT100 Offset,PR[24:Rotate_Offset] ;
4811:L P[3134]  R[157] mm/sec CNT100 Offset,PR[24:Rotate_Offset] ;
4812:L P[3135]  R[157] mm/sec CNT100 Offset,PR[24:Rotate_Offset] ;
4813:L P[3136]  R[157] mm/sec CNT100 Offset,PR[24:Rotate_Offset] ;
4814:L P[3137]  R[157] mm/sec CNT100 Offset,PR[24:Rotate_Offset] ;
4815:L P[3138]  R[157] mm/sec CNT100 Offset,PR[24:Rotate_Offset] ;
4816:L P[3139]  R[157] mm/sec CNT100 Offset,PR[24:Rotate_Offset] ;
4817:L P[3140]  R[157] mm/sec CNT100 Offset,PR[24:Rotate_Offset] ;
4818:L P[3141]  R[157] mm/sec CNT100 TA    0.00sec,CALL RUN_LASER_STOP Offset,PR[26:Stop_Offset] ;
4820:L P[3141]  R[157] mm/sec FINE Offset,PR[76:Offst_dprt] ;
4821:L P[3142]  R[157] mm/sec CNT100 Offset,PR[24:Rotate_Offset] ;
4822:L P[3143]  R[157] mm/sec CNT100 Offset,PR[24:Rotate_Offset] ;
4823:L P[3144]  R[157] mm/sec CNT100 Offset,PR[24:Rotate_Offset] ;
4824:L P[3145]  R[157] mm/sec CNT100 Offset,PR[24:Rotate_Offset] ;
4825:L P[3146]  R[157] mm/sec CNT100 Offset,PR[24:Rotate_Offset] ;
4826:L P[3147]  R[157] mm/sec CNT100 Offset,PR[24:Rotate_Offset] ;
4827: !Pass239 ;
4828: LBL[1239:Pass239] ;
4829:L P[3148]  R[157] mm/sec FINE Offset,PR[78:Offst_apprch]  ;
4830: WAIT   0.20(sec) ;
4831:L P[3148]  R[157] mm/sec CNT100 TA    0.00sec,CALL RUN_LASER_START Offset,PR[25:Start_Offset] ;
4833:L P[3149]  R[157] mm/sec CNT100 Offset,PR[24:Rotate_Offset] ;
4834:L P[3150]  R[157] mm/sec CNT100 Offset,PR[24:Rotate_Offset] ;
4835:L P[3151]  R[157] mm/sec CNT100 Offset,PR[24:Rotate_Offset] ;
4836:L P[3152]  R[157] mm/sec CNT100 Offset,PR[24:Rotate_Offset] ;
4837:L P[3153]  R[157] mm/sec CNT100 Offset,PR[24:Rotate_Offset] ;
4838:L P[3154]  R[157] mm/sec CNT100 Offset,PR[24:Rotate_Offset] ;
4839:L P[3155]  R[157] mm/sec CNT100 Offset,PR[24:Rotate_Offset] ;
4840:L P[3156]  R[157] mm/sec CNT100 Offset,PR[24:Rotate_Offset] ;
4841:L P[3157]  R[157] mm/sec CNT100 Offset,PR[24:Rotate_Offset] ;
4842:L P[3158]  R[157] mm/sec CNT100 Offset,PR[24:Rotate_Offset] ;
4843:L P[3159]  R[157] mm/sec CNT100 Offset,PR[24:Rotate_Offset] ;
4844:L P[3160]  R[157] mm/sec CNT100 Offset,PR[24:Rotate_Offset] ;
4845:L P[3161]  R[157] mm/sec CNT100 Offset,PR[24:Rotate_Offset] ;
4846:L P[3162]  R[157] mm/sec CNT100 Offset,PR[24:Rotate_Offset] ;
4847:L P[3163]  R[157] mm/sec CNT100 Offset,PR[24:Rotate_Offset] ;
4848:L P[3164]  R[157] mm/sec CNT100 Offset,PR[24:Rotate_Offset] ;
4849:L P[3165]  R[157] mm/sec CNT100 Offset,PR[24:Rotate_Offset] ;
4850:L P[3166]  R[157] mm/sec CNT100 Offset,PR[24:Rotate_Offset] ;
4851:L P[3167]  R[157] mm/sec CNT100 Offset,PR[24:Rotate_Offset] ;
4852:L P[3168]  R[157] mm/sec CNT100 Offset,PR[24:Rotate_Offset] ;
4853:L P[3169]  R[157] mm/sec CNT100 Offset,PR[24:Rotate_Offset] ;
4854:L P[3170]  R[157] mm/sec CNT100 Offset,PR[24:Rotate_Offset] ;
4855:L P[3171]  R[157] mm/sec CNT100 Offset,PR[24:Rotate_Offset] ;
4856:L P[3172]  R[157] mm/sec CNT100 Offset,PR[24:Rotate_Offset] ;
4857:L P[3173]  R[157] mm/sec CNT100 Offset,PR[24:Rotate_Offset] ;
4858:L P[3174]  R[157] mm/sec CNT100 Offset,PR[24:Rotate_Offset] ;
4859:L P[3175]  R[157] mm/sec CNT100 Offset,PR[24:Rotate_Offset] ;
4860:L P[3176]  R[157] mm/sec CNT100 Offset,PR[24:Rotate_Offset] ;
4861:L P[3177]  R[157] mm/sec CNT100 Offset,PR[24:Rotate_Offset] ;
4862:L P[3178]  R[157] mm/sec CNT100 Offset,PR[24:Rotate_Offset] ;
4863:L P[3179]  R[157] mm/sec CNT100 Offset,PR[24:Rotate_Offset] ;
4864:L P[3180]  R[157] mm/sec CNT100 Offset,PR[24:Rotate_Offset] ;
4865:L P[3181]  R[157] mm/sec CNT100 Offset,PR[24:Rotate_Offset] ;
4866:L P[3182]  R[157] mm/sec CNT100 Offset,PR[24:Rotate_Offset] ;
4867:L P[3183]  R[157] mm/sec CNT100 Offset,PR[24:Rotate_Offset] ;
4868:L P[3184]  R[157] mm/sec CNT100 Offset,PR[24:Rotate_Offset] ;
4869:L P[3185]  R[157] mm/sec CNT100 Offset,PR[24:Rotate_Offset] ;
4870:L P[3186]  R[157] mm/sec CNT100 Offset,PR[24:Rotate_Offset] ;
4871:L P[3187]  R[157] mm/sec CNT100 Offset,PR[24:Rotate_Offset] ;
4872:L P[3188]  R[157] mm/sec CNT100 Offset,PR[24:Rotate_Offset] ;
4873:L P[3189]  R[157] mm/sec CNT100 Offset,PR[24:Rotate_Offset] ;
4874:L P[3190]  R[157] mm/sec CNT100 Offset,PR[24:Rotate_Offset] ;
4875:L P[3191]  R[157] mm/sec CNT100 Offset,PR[24:Rotate_Offset] ;
4876:L P[3192]  R[157] mm/sec CNT100 Offset,PR[24:Rotate_Offset] ;
4877:L P[3193]  R[157] mm/sec CNT100 Offset,PR[24:Rotate_Offset] ;
4878:L P[3194]  R[157] mm/sec CNT100 Offset,PR[24:Rotate_Offset] ;
4879:L P[3195]  R[157] mm/sec CNT100 Offset,PR[24:Rotate_Offset] ;
4880:L P[3196]  R[157] mm/sec CNT100 Offset,PR[24:Rotate_Offset] ;
4881:L P[3197]  R[157] mm/sec CNT100 TA    0.00sec,CALL RUN_LASER_STOP Offset,PR[26:Stop_Offset] ;
4883:L P[3197]  R[157] mm/sec FINE Offset,PR[76:Offst_dprt] ;
4884:L P[3198]  R[157] mm/sec CNT100 Offset,PR[24:Rotate_Offset] ;
4885:L P[3199]  R[157] mm/sec CNT100 Offset,PR[24:Rotate_Offset] ;
4886:L P[3200]  R[157] mm/sec CNT100 Offset,PR[24:Rotate_Offset] ;
4887:L P[3201]  R[157] mm/sec CNT100 Offset,PR[24:Rotate_Offset] ;
4888:L P[3202]  R[157] mm/sec CNT100 Offset,PR[24:Rotate_Offset] ;
4889:L P[3203]  R[157] mm/sec CNT100 Offset,PR[24:Rotate_Offset] ;
4890: !Pass240 ;
4891: LBL[1240:Pass240] ;
4892:L P[3204]  R[157] mm/sec FINE Offset,PR[78:Offst_apprch]  ;
4893: WAIT   0.20(sec) ;
4894:L P[3204]  R[157] mm/sec CNT100 TA    0.00sec,CALL RUN_LASER_START Offset,PR[25:Start_Offset] ;
4896:L P[3205]  R[157] mm/sec CNT100 Offset,PR[24:Rotate_Offset] ;
4897:L P[3206]  R[157] mm/sec CNT100 Offset,PR[24:Rotate_Offset] ;
4898:L P[3207]  R[157] mm/sec CNT100 Offset,PR[24:Rotate_Offset] ;
4899:L P[3208]  R[157] mm/sec CNT100 Offset,PR[24:Rotate_Offset] ;
4900:L P[3209]  R[157] mm/sec CNT100 Offset,PR[24:Rotate_Offset] ;
4901:L P[3210]  R[157] mm/sec CNT100 Offset,PR[24:Rotate_Offset] ;
4902:L P[3211]  R[157] mm/sec CNT100 Offset,PR[24:Rotate_Offset] ;
4903:L P[3212]  R[157] mm/sec CNT100 Offset,PR[24:Rotate_Offset] ;
4904:L P[3213]  R[157] mm/sec CNT100 Offset,PR[24:Rotate_Offset] ;
4905:L P[3214]  R[157] mm/sec CNT100 Offset,PR[24:Rotate_Offset] ;
4906:L P[3215]  R[157] mm/sec CNT100 Offset,PR[24:Rotate_Offset] ;
4907:L P[3216]  R[157] mm/sec CNT100 Offset,PR[24:Rotate_Offset] ;
4908:L P[3217]  R[157] mm/sec CNT100 Offset,PR[24:Rotate_Offset] ;
4909:L P[3218]  R[157] mm/sec CNT100 Offset,PR[24:Rotate_Offset] ;
4910:L P[3219]  R[157] mm/sec CNT100 Offset,PR[24:Rotate_Offset] ;
4911:L P[3220]  R[157] mm/sec CNT100 Offset,PR[24:Rotate_Offset] ;
4912:L P[3221]  R[157] mm/sec CNT100 Offset,PR[24:Rotate_Offset] ;
4913:L P[3222]  R[157] mm/sec CNT100 Offset,PR[24:Rotate_Offset] ;
4914:L P[3223]  R[157] mm/sec CNT100 Offset,PR[24:Rotate_Offset] ;
4915:L P[3224]  R[157] mm/sec CNT100 Offset,PR[24:Rotate_Offset] ;
4916:L P[3225]  R[157] mm/sec CNT100 Offset,PR[24:Rotate_Offset] ;
4917:L P[3226]  R[157] mm/sec CNT100 Offset,PR[24:Rotate_Offset] ;
4918:L P[3227]  R[157] mm/sec CNT100 Offset,PR[24:Rotate_Offset] ;
4919:L P[3228]  R[157] mm/sec CNT100 Offset,PR[24:Rotate_Offset] ;
4920:L P[3229]  R[157] mm/sec CNT100 Offset,PR[24:Rotate_Offset] ;
4921:L P[3230]  R[157] mm/sec CNT100 Offset,PR[24:Rotate_Offset] ;
4922:L P[3231]  R[157] mm/sec CNT100 Offset,PR[24:Rotate_Offset] ;
4923:L P[3232]  R[157] mm/sec CNT100 Offset,PR[24:Rotate_Offset] ;
4924:L P[3233]  R[157] mm/sec CNT100 Offset,PR[24:Rotate_Offset] ;
4925:L P[3234]  R[157] mm/sec CNT100 Offset,PR[24:Rotate_Offset] ;
4926:L P[3235]  R[157] mm/sec CNT100 Offset,PR[24:Rotate_Offset] ;
4927:L P[3236]  R[157] mm/sec CNT100 Offset,PR[24:Rotate_Offset] ;
4928:L P[3237]  R[157] mm/sec CNT100 Offset,PR[24:Rotate_Offset] ;
4929:L P[3238]  R[157] mm/sec CNT100 Offset,PR[24:Rotate_Offset] ;
4930:L P[3239]  R[157] mm/sec CNT100 Offset,PR[24:Rotate_Offset] ;
4931:L P[3240]  R[157] mm/sec CNT100 Offset,PR[24:Rotate_Offset] ;
4932:L P[3241]  R[157] mm/sec CNT100 Offset,PR[24:Rotate_Offset] ;
4933:L P[3242]  R[157] mm/sec CNT100 Offset,PR[24:Rotate_Offset] ;
4934:L P[3243]  R[157] mm/sec CNT100 Offset,PR[24:Rotate_Offset] ;
4935:L P[3244]  R[157] mm/sec CNT100 Offset,PR[24:Rotate_Offset] ;
4936:L P[3245]  R[157] mm/sec CNT100 Offset,PR[24:Rotate_Offset] ;
4937:L P[3246]  R[157] mm/sec CNT100 Offset,PR[24:Rotate_Offset] ;
4938:L P[3247]  R[157] mm/sec CNT100 Offset,PR[24:Rotate_Offset] ;
4939:L P[3248]  R[157] mm/sec CNT100 Offset,PR[24:Rotate_Offset] ;
4940:L P[3249]  R[157] mm/sec CNT100 Offset,PR[24:Rotate_Offset] ;
4941:L P[3250]  R[157] mm/sec CNT100 Offset,PR[24:Rotate_Offset] ;
4942:L P[3251]  R[157] mm/sec CNT100 Offset,PR[24:Rotate_Offset] ;
4943:L P[3252]  R[157] mm/sec CNT100 TA    0.00sec,CALL RUN_LASER_STOP Offset,PR[26:Stop_Offset] ;
4945:L P[3252]  R[157] mm/sec FINE Offset,PR[76:Offst_dprt] ;
4946:L P[3253]  R[157] mm/sec CNT100 Offset,PR[24:Rotate_Offset] ;
4947:L P[3254]  R[157] mm/sec CNT100 Offset,PR[24:Rotate_Offset] ;
4948:L P[3255]  R[157] mm/sec CNT100 Offset,PR[24:Rotate_Offset] ;
4949:L P[3256]  R[157] mm/sec CNT100 Offset,PR[24:Rotate_Offset] ;
4950:L P[3257]  R[157] mm/sec CNT100 Offset,PR[24:Rotate_Offset] ;
4951:L P[3258]  R[157] mm/sec CNT100 Offset,PR[24:Rotate_Offset] ;
4952: !Pass241 ;
4953: LBL[1241:Pass241] ;
4954:L P[3259]  R[157] mm/sec FINE Offset,PR[78:Offst_apprch]  ;
4955: WAIT   0.20(sec) ;
4956:L P[3259]  R[157] mm/sec CNT100 TA    0.00sec,CALL RUN_LASER_START Offset,PR[25:Start_Offset] ;
4958:L P[3260]  R[157] mm/sec CNT100 Offset,PR[24:Rotate_Offset] ;
4959:L P[3261]  R[157] mm/sec CNT100 Offset,PR[24:Rotate_Offset] ;
4960:L P[3262]  R[157] mm/sec CNT100 Offset,PR[24:Rotate_Offset] ;
4961:L P[3263]  R[157] mm/sec CNT100 Offset,PR[24:Rotate_Offset] ;
4962:L P[3264]  R[157] mm/sec CNT100 Offset,PR[24:Rotate_Offset] ;
4963:L P[3265]  R[157] mm/sec CNT100 Offset,PR[24:Rotate_Offset] ;
4964:L P[3266]  R[157] mm/sec CNT100 Offset,PR[24:Rotate_Offset] ;
4965:L P[3267]  R[157] mm/sec CNT100 Offset,PR[24:Rotate_Offset] ;
4966:L P[3268]  R[157] mm/sec CNT100 Offset,PR[24:Rotate_Offset] ;
4967:L P[3269]  R[157] mm/sec CNT100 Offset,PR[24:Rotate_Offset] ;
4968:L P[3270]  R[157] mm/sec CNT100 Offset,PR[24:Rotate_Offset] ;
4969:L P[3271]  R[157] mm/sec CNT100 Offset,PR[24:Rotate_Offset] ;
4970:L P[3272]  R[157] mm/sec CNT100 Offset,PR[24:Rotate_Offset] ;
4971:L P[3273]  R[157] mm/sec CNT100 Offset,PR[24:Rotate_Offset] ;
4972:L P[3274]  R[157] mm/sec CNT100 Offset,PR[24:Rotate_Offset] ;
4973:L P[3275]  R[157] mm/sec CNT100 Offset,PR[24:Rotate_Offset] ;
4974:L P[3276]  R[157] mm/sec CNT100 Offset,PR[24:Rotate_Offset] ;
4975:L P[3277]  R[157] mm/sec CNT100 Offset,PR[24:Rotate_Offset] ;
4976:L P[3278]  R[157] mm/sec CNT100 Offset,PR[24:Rotate_Offset] ;
4977:L P[3279]  R[157] mm/sec CNT100 Offset,PR[24:Rotate_Offset] ;
4978:L P[3280]  R[157] mm/sec CNT100 Offset,PR[24:Rotate_Offset] ;
4979:L P[3281]  R[157] mm/sec CNT100 Offset,PR[24:Rotate_Offset] ;
4980:L P[3282]  R[157] mm/sec CNT100 Offset,PR[24:Rotate_Offset] ;
4981:L P[3283]  R[157] mm/sec CNT100 Offset,PR[24:Rotate_Offset] ;
4982:L P[3284]  R[157] mm/sec CNT100 Offset,PR[24:Rotate_Offset] ;
4983:L P[3285]  R[157] mm/sec CNT100 Offset,PR[24:Rotate_Offset] ;
4984:L P[3286]  R[157] mm/sec CNT100 Offset,PR[24:Rotate_Offset] ;
4985:L P[3287]  R[157] mm/sec CNT100 Offset,PR[24:Rotate_Offset] ;
4986:L P[3288]  R[157] mm/sec CNT100 Offset,PR[24:Rotate_Offset] ;
4987:L P[3289]  R[157] mm/sec CNT100 Offset,PR[24:Rotate_Offset] ;
4988:L P[3290]  R[157] mm/sec CNT100 Offset,PR[24:Rotate_Offset] ;
4989:L P[3291]  R[157] mm/sec CNT100 Offset,PR[24:Rotate_Offset] ;
4990:L P[3292]  R[157] mm/sec CNT100 Offset,PR[24:Rotate_Offset] ;
4991:L P[3293]  R[157] mm/sec CNT100 Offset,PR[24:Rotate_Offset] ;
4992:L P[3294]  R[157] mm/sec CNT100 Offset,PR[24:Rotate_Offset] ;
4993:L P[3295]  R[157] mm/sec CNT100 Offset,PR[24:Rotate_Offset] ;
4994:L P[3296]  R[157] mm/sec CNT100 Offset,PR[24:Rotate_Offset] ;
4995:L P[3297]  R[157] mm/sec CNT100 Offset,PR[24:Rotate_Offset] ;
4996:L P[3298]  R[157] mm/sec CNT100 Offset,PR[24:Rotate_Offset] ;
4997:L P[3299]  R[157] mm/sec CNT100 Offset,PR[24:Rotate_Offset] ;
4998:L P[3300]  R[157] mm/sec CNT100 Offset,PR[24:Rotate_Offset] ;
4999:L P[3301]  R[157] mm/sec CNT100 Offset,PR[24:Rotate_Offset] ;
5000:L P[3302]  R[157] mm/sec CNT100 Offset,PR[24:Rotate_Offset] ;
5001:L P[3303]  R[157] mm/sec CNT100 Offset,PR[24:Rotate_Offset] ;
5002:L P[3304]  R[157] mm/sec CNT100 Offset,PR[24:Rotate_Offset] ;
5003:L P[3305]  R[157] mm/sec CNT100 Offset,PR[24:Rotate_Offset] ;
5004:L P[3306]  R[157] mm/sec CNT100 TA    0.00sec,CALL RUN_LASER_STOP Offset,PR[26:Stop_Offset] ;
5006:L P[3306]  R[157] mm/sec FINE Offset,PR[76:Offst_dprt] ;
5007:L P[3307]  R[157] mm/sec CNT100 Offset,PR[24:Rotate_Offset] ;
5008:L P[3308]  R[157] mm/sec CNT100 Offset,PR[24:Rotate_Offset] ;
5009:L P[3309]  R[157] mm/sec CNT100 Offset,PR[24:Rotate_Offset] ;
5010: ;
5011: ! Home ;
5012: ;
5013:J P[3310]  R[225] % FINE ;
5014: LBL[8999:EOF];
/POS
P[1]{
   GP1:
	UF : 7, UT : 3,
	J1 =  -129.583 deg,	J2 =    24.319 deg,	J3 =   -28.425 deg,
	J4 =   110.695 deg,	J5 =   124.219 deg,	J6 =   -55.036 deg
};
P[2]{
   GP1:
	UF : 7, UT : 3,	CONFIG : 'F U T, 0, 1, 0',
	X =  -392.700  mm,	Y =     0.000  mm,	Z =     0.000  mm,
	W =  -167.363 deg,	P =     0.001 deg,	R =   -75.580 deg
};
P[3]{
   GP1:
	UF : 7, UT : 3,	CONFIG : 'F U T, 0, 1, 0',
	X =  -392.700  mm,	Y =     0.000  mm,	Z =     0.000  mm,
	W =  -167.363 deg,	P =     0.001 deg,	R =   -75.580 deg
};
P[4]{
   GP1:
	UF : 7, UT : 3,	CONFIG : 'F U T, 0, 1, 0',
	X =  -392.700  mm,	Y =     0.000  mm,	Z =     0.000  mm,
	W =  -167.363 deg,	P =     0.001 deg,	R =   -75.580 deg
};
P[5]{
   GP1:
	UF : 7, UT : 3,	CONFIG : 'F U T, 0, 1, 0',
	X =  -392.700  mm,	Y =     0.000  mm,	Z =     0.000  mm,
	W =  -167.363 deg,	P =     0.001 deg,	R =   -75.580 deg
};
P[6]{
   GP1:
	UF : 7, UT : 3,	CONFIG : 'F U T, 0, 1, 0',
	X =  -391.802  mm,	Y =    26.450  mm,	Z =     0.000  mm,
	W =  -167.331 deg,	P =    -0.011 deg,	R =   -78.833 deg
};
P[7]{
   GP1:
	UF : 7, UT : 3,	CONFIG : 'F U T, 0, 1, 0',
	X =  -389.578  mm,	Y =    49.276  mm,	Z =     0.001  mm,
	W =  -167.302 deg,	P =    -0.017 deg,	R =   -82.117 deg
};
P[8]{
   GP1:
	UF : 7, UT : 3,	CONFIG : 'F U T, 0, 0, 0',
	X =  -386.090  mm,	Y =    71.652  mm,	Z =     0.002  mm,
	W =  -167.272 deg,	P =    -0.020 deg,	R =   -85.505 deg
};
P[9]{
   GP1:
	UF : 7, UT : 3,	CONFIG : 'F U T, 0, 0, 0',
	X =  -381.740  mm,	Y =    92.040  mm,	Z =     0.005  mm,
	W =  -167.115 deg,	P =    -0.053 deg,	R =   -88.368 deg
};
P[10]{
   GP1:
	UF : 7, UT : 3,	CONFIG : 'F U T, 0, 0, 0',
	X =  -375.752  mm,	Y =   114.056  mm,	Z =     0.017  mm,
	W =  -166.473 deg,	P =    -0.189 deg,	R =   -91.893 deg
};
P[11]{
   GP1:
	UF : 7, UT : 3,	CONFIG : 'F U T, 0, 0, 0',
	X =  -372.289  mm,	Y =   124.892  mm,	Z =     0.028  mm,
	W =  -165.851 deg,	P =    -0.342 deg,	R =   -93.426 deg
};
P[12]{
   GP1:
	UF : 7, UT : 3,	CONFIG : 'F U T, 0, 0, 0',
	X =  -366.899  mm,	Y =   139.931  mm,	Z =     0.050  mm,
	W =  -164.775 deg,	P =    -0.619 deg,	R =   -95.793 deg
};
P[13]{
   GP1:
	UF : 7, UT : 3,	CONFIG : 'F U T, 0, 0, 0',
	X =  -361.833  mm,	Y =   152.613  mm,	Z =     0.066  mm,
	W =  -163.795 deg,	P =    -0.891 deg,	R =   -97.858 deg
};
P[14]{
   GP1:
	UF : 7, UT : 3,	CONFIG : 'F U T, 0, 0, 0',
	X =  -356.336  mm,	Y =   164.995  mm,	Z =     0.078  mm,
	W =  -163.250 deg,	P =    -1.098 deg,	R =   -99.819 deg
};
P[15]{
   GP1:
	UF : 7, UT : 3,	CONFIG : 'F U T, 0, 0, 0',
	X =  -354.115  mm,	Y =   169.721  mm,	Z =     0.076  mm,
	W =  -163.289 deg,	P =    -1.119 deg,	R =  -100.688 deg
};
P[16]{
   GP1:
	UF : 7, UT : 3,	CONFIG : 'F U T, 0, 0, 0',
	X =  -349.006  mm,	Y =   179.976  mm,	Z =     0.062  mm,
	W =  -164.035 deg,	P =    -0.997 deg,	R =  -102.257 deg
};
P[17]{
   GP1:
	UF : 7, UT : 3,	CONFIG : 'F U T, 0, 0, 0',
	X =  -340.090  mm,	Y =   196.308  mm,	Z =     0.033  mm,
	W =  -165.623 deg,	P =    -0.542 deg,	R =  -104.913 deg
};
P[18]{
   GP1:
	UF : 7, UT : 3,	CONFIG : 'F U T, 0, 0, 0',
	X =  -329.378  mm,	Y =   213.813  mm,	Z =     0.015  mm,
	W =  -166.590 deg,	P =    -0.241 deg,	R =  -107.947 deg
};
P[19]{
   GP1:
	UF : 7, UT : 3,	CONFIG : 'F U T, 0, 0, 0',
	X =  -322.013  mm,	Y =   224.727  mm,	Z =     0.009  mm,
	W =  -166.893 deg,	P =    -0.146 deg,	R =  -109.790 deg
};
P[20]{
   GP1:
	UF : 7, UT : 3,	CONFIG : 'F U T, 0, 0, 0',
	X =  -310.542  mm,	Y =   240.344  mm,	Z =     0.005  mm,
	W =  -167.112 deg,	P =    -0.076 deg,	R =  -112.590 deg
};
P[21]{
   GP1:
	UF : 7, UT : 3,	CONFIG : 'F U T, 0, 0, 0',
	X =  -298.316  mm,	Y =   255.379  mm,	Z =     0.003  mm,
	W =  -167.176 deg,	P =    -0.052 deg,	R =  -115.513 deg
};
P[22]{
   GP1:
	UF : 7, UT : 3,	CONFIG : 'F U T, 0, 0, 0',
	X =  -285.356  mm,	Y =   269.764  mm,	Z =     0.002  mm,
	W =  -167.241 deg,	P =    -0.034 deg,	R =  -118.438 deg
};
P[23]{
   GP1:
	UF : 7, UT : 3,	CONFIG : 'F U T, 0, 0, 0',
	X =  -267.605  mm,	Y =   287.387  mm,	Z =     0.002  mm,
	W =  -167.262 deg,	P =    -0.022 deg,	R =  -122.038 deg
};
P[24]{
   GP1:
	UF : 7, UT : 3,	CONFIG : 'F U T, 0, 0, 0',
	X =  -248.465  mm,	Y =   304.100  mm,	Z =     0.001  mm,
	W =  -167.285 deg,	P =    -0.013 deg,	R =  -125.703 deg
};
P[25]{
   GP1:
	UF : 7, UT : 3,	CONFIG : 'F U T, 0, 0, 0',
	X =  -228.526  mm,	Y =   319.349  mm,	Z =     0.001  mm,
	W =  -167.307 deg,	P =    -0.007 deg,	R =  -129.326 deg
};
P[26]{
   GP1:
	UF : 7, UT : 3,	CONFIG : 'F U T, 0, 0, 0',
	X =  -207.697  mm,	Y =   333.268  mm,	Z =     0.000  mm,
	W =  -167.331 deg,	P =    -0.003 deg,	R =  -132.943 deg
};
P[27]{
   GP1:
	UF : 7, UT : 3,	CONFIG : 'F U T, 0, 0, 0',
	X =  -186.179  mm,	Y =   345.739  mm,	Z =     0.000  mm,
	W =  -167.354 deg,	P =    -0.003 deg,	R =  -136.585 deg
};
P[28]{
   GP1:
	UF : 7, UT : 3,	CONFIG : 'F U T, 0, 0, 0',
	X =  -163.790  mm,	Y =   356.887  mm,	Z =     0.000  mm,
	W =  -167.354 deg,	P =    -0.002 deg,	R =  -140.267 deg
};
P[29]{
   GP1:
	UF : 7, UT : 3,	CONFIG : 'F U T, 0, 0, 0',
	X =  -140.820  mm,	Y =   366.558  mm,	Z =     0.000  mm,
	W =  -167.354 deg,	P =    -0.002 deg,	R =  -144.004 deg
};
P[30]{
   GP1:
	UF : 7, UT : 3,	CONFIG : 'F U T, 0, 0, 0',
	X =  -117.155  mm,	Y =   374.796  mm,	Z =     0.000  mm,
	W =  -167.354 deg,	P =    -0.001 deg,	R =  -147.677 deg
};
P[31]{
   GP1:
	UF : 7, UT : 3,	CONFIG : 'F U T, 0, 0, 0',
	X =   -92.957  mm,	Y =   381.524  mm,	Z =     0.000  mm,
	W =  -167.355 deg,	P =     0.000 deg,	R =  -151.341 deg
};
P[32]{
   GP1:
	UF : 7, UT : 3,	CONFIG : 'F U T, 0, 0, 0',
	X =   -68.192  mm,	Y =   386.720  mm,	Z =     0.000  mm,
	W =  -167.355 deg,	P =     0.000 deg,	R =  -154.997 deg
};
P[33]{
   GP1:
	UF : 7, UT : 3,	CONFIG : 'F U T, 0, 0, 0',
	X =   -43.073  mm,	Y =   390.318  mm,	Z =     0.000  mm,
	W =  -167.355 deg,	P =     0.001 deg,	R =  -158.672 deg
};
P[34]{
   GP1:
	UF : 7, UT : 3,	CONFIG : 'F U T, 0, 0, 0',
	X =   -17.715  mm,	Y =   392.287  mm,	Z =     0.000  mm,
	W =  -167.356 deg,	P =     0.001 deg,	R =  -162.341 deg
};
P[35]{
   GP1:
	UF : 7, UT : 3,	CONFIG : 'F U T, 0, 0, 0',
	X =     7.756  mm,	Y =   392.610  mm,	Z =     0.000  mm,
	W =  -167.356 deg,	P =     0.002 deg,	R =  -166.029 deg
};
P[36]{
   GP1:
	UF : 7, UT : 3,	CONFIG : 'F U T, 0, 0, 0',
	X =    33.030  mm,	Y =   391.294  mm,	Z =     0.000  mm,
	W =  -167.356 deg,	P =     0.002 deg,	R =  -169.679 deg
};
P[37]{
   GP1:
	UF : 7, UT : 3,	CONFIG : 'F U T, 0, 0, 0',
	X =    57.922  mm,	Y =   388.384  mm,	Z =     0.000  mm,
	W =  -167.357 deg,	P =     0.002 deg,	R =  -173.353 deg
};
P[38]{
   GP1:
	UF : 7, UT : 3,	CONFIG : 'F U T, 0, 0, 0',
	X =    82.591  mm,	Y =   383.893  mm,	Z =     0.000  mm,
	W =  -167.357 deg,	P =     0.003 deg,	R =  -177.012 deg
};
P[39]{
   GP1:
	UF : 7, UT : 3,	CONFIG : 'F U T, 0, 0, 0',
	X =   106.804  mm,	Y =   377.873  mm,	Z =     0.000  mm,
	W =  -167.358 deg,	P =     0.003 deg,	R =   179.274 deg
};
P[40]{
   GP1:
	UF : 7, UT : 3,	CONFIG : 'F U T, 0, 0, 0',
	X =   130.591  mm,	Y =   370.330  mm,	Z =     0.000  mm,
	W =  -167.358 deg,	P =     0.003 deg,	R =   175.574 deg
};
P[41]{
   GP1:
	UF : 7, UT : 3,	CONFIG : 'F U T, 0, 0, 0',
	X =   154.020  mm,	Y =   361.222  mm,	Z =     0.000  mm,
	W =  -167.359 deg,	P =     0.003 deg,	R =   171.885 deg
};
P[42]{
   GP1:
	UF : 7, UT : 3,	CONFIG : 'F U T, 0, 0, 0',
	X =   176.898  mm,	Y =   350.590  mm,	Z =     0.000  mm,
	W =  -167.359 deg,	P =     0.003 deg,	R =   168.224 deg
};
P[43]{
   GP1:
	UF : 7, UT : 3,	CONFIG : 'F U T, 0, 0, 0',
	X =   199.109  mm,	Y =   338.469  mm,	Z =     0.000  mm,
	W =  -167.360 deg,	P =     0.003 deg,	R =   164.571 deg
};
P[44]{
   GP1:
	UF : 7, UT : 3,	CONFIG : 'F U T, 0, 0, 0',
	X =   220.586  mm,	Y =   324.878  mm,	Z =     0.000  mm,
	W =  -167.360 deg,	P =     0.003 deg,	R =   160.893 deg
};
P[45]{
   GP1:
	UF : 7, UT : 3,	CONFIG : 'F U T, 0, 0, 0',
	X =   241.190  mm,	Y =   309.887  mm,	Z =     0.000  mm,
	W =  -167.361 deg,	P =     0.003 deg,	R =   157.223 deg
};
P[46]{
   GP1:
	UF : 7, UT : 3,	CONFIG : 'F U T, 0, 0, 0',
	X =   260.831  mm,	Y =   293.544  mm,	Z =     0.000  mm,
	W =  -167.361 deg,	P =     0.003 deg,	R =   153.513 deg
};
P[47]{
   GP1:
	UF : 7, UT : 3,	CONFIG : 'F U T, 0, 0, 0',
	X =   279.253  mm,	Y =   276.075  mm,	Z =     0.000  mm,
	W =  -167.361 deg,	P =     0.003 deg,	R =   149.836 deg
};
P[48]{
   GP1:
	UF : 7, UT : 3,	CONFIG : 'F U T, 0, 0, 0',
	X =   296.378  mm,	Y =   257.597  mm,	Z =     0.000  mm,
	W =  -167.362 deg,	P =     0.003 deg,	R =   146.173 deg
};
P[49]{
   GP1:
	UF : 7, UT : 3,	CONFIG : 'F U T, 0, 0, 0',
	X =   312.233  mm,	Y =   238.128  mm,	Z =     0.000  mm,
	W =  -167.362 deg,	P =     0.003 deg,	R =   142.483 deg
};
P[50]{
   GP1:
	UF : 7, UT : 3,	CONFIG : 'F U T, 0, 0, 0',
	X =   326.797  mm,	Y =   217.714  mm,	Z =     0.000  mm,
	W =  -167.362 deg,	P =     0.003 deg,	R =   138.727 deg
};
P[51]{
   GP1:
	UF : 7, UT : 3,	CONFIG : 'F U T, 0, 0, 0',
	X =   339.960  mm,	Y =   196.538  mm,	Z =     0.000  mm,
	W =  -167.363 deg,	P =     0.002 deg,	R =   135.023 deg
};
P[52]{
   GP1:
	UF : 7, UT : 3,	CONFIG : 'F U T, 0, 0, 0',
	X =   351.889  mm,	Y =   174.294  mm,	Z =     0.000  mm,
	W =  -167.363 deg,	P =     0.002 deg,	R =   131.327 deg
};
P[53]{
   GP1:
	UF : 7, UT : 3,	CONFIG : 'F U T, 0, 0, 0',
	X =   362.374  mm,	Y =   151.302  mm,	Z =     0.000  mm,
	W =  -167.363 deg,	P =     0.002 deg,	R =   127.655 deg
};
P[54]{
   GP1:
	UF : 7, UT : 3,	CONFIG : 'F U T, 0, 0, 0',
	X =   371.395  mm,	Y =   127.559  mm,	Z =     0.000  mm,
	W =  -167.363 deg,	P =     0.002 deg,	R =   123.988 deg
};
P[55]{
   GP1:
	UF : 7, UT : 3,	CONFIG : 'F U T, 0, 0, 0',
	X =   378.856  mm,	Y =   103.309  mm,	Z =     0.000  mm,
	W =  -167.363 deg,	P =     0.001 deg,	R =   120.320 deg
};
P[56]{
   GP1:
	UF : 7, UT : 3,	CONFIG : 'F U T, 0, 0, 0',
	X =   384.730  mm,	Y =    78.643  mm,	Z =     0.000  mm,
	W =  -167.363 deg,	P =     0.001 deg,	R =   116.658 deg
};
P[57]{
   GP1:
	UF : 7, UT : 3,	CONFIG : 'F U T, 0, 0, 0',
	X =   389.009  mm,	Y =    53.590  mm,	Z =     0.000  mm,
	W =  -167.364 deg,	P =     0.001 deg,	R =   112.982 deg
};
P[58]{
   GP1:
	UF : 7, UT : 3,	CONFIG : 'F U T, 0, 0, 0',
	X =   391.646  mm,	Y =    28.482  mm,	Z =     0.000  mm,
	W =  -167.364 deg,	P =     0.000 deg,	R =   109.349 deg
};
P[59]{
   GP1:
	UF : 7, UT : 3,	CONFIG : 'F U T, 0, 0, 0',
	X =   392.700  mm,	Y =     0.000  mm,	Z =     0.000  mm,
	W =  -167.363 deg,	P =     0.000 deg,	R =   105.687 deg
};
P[60]{
   GP1:
	UF : 7, UT : 3,	CONFIG : 'F U T, 0, 0, 0',
	X =   392.700  mm,	Y =     0.000  mm,	Z =     0.000  mm,
	W =  -167.363 deg,	P =     0.000 deg,	R =   105.687 deg
};
P[61]{
   GP1:
	UF : 7, UT : 3,	CONFIG : 'F U T, 0, 0, 0',
	X =   392.700  mm,	Y =     0.000  mm,	Z =     0.000  mm,
	W =  -167.363 deg,	P =     0.000 deg,	R =   105.687 deg
};
P[62]{
   GP1:
	UF : 7, UT : 3,	CONFIG : 'F U T, 0, 0, 0',
	X =   392.700  mm,	Y =     0.000  mm,	Z =     0.000  mm,
	W =  -167.363 deg,	P =     0.000 deg,	R =   105.687 deg
};
P[63]{
   GP1:
	UF : 7, UT : 3,	CONFIG : 'F U T, 0, 0, 0',
	X =   389.566  mm,	Y =     0.000  mm,	Z =     0.000  mm,
	W =  -167.363 deg,	P =     0.000 deg,	R =   105.687 deg
};
P[64]{
   GP1:
	UF : 7, UT : 3,	CONFIG : 'F U T, 0, 0, 0',
	X =   389.566  mm,	Y =     0.000  mm,	Z =     0.000  mm,
	W =  -167.363 deg,	P =     0.000 deg,	R =   105.687 deg
};
P[65]{
   GP1:
	UF : 7, UT : 3,	CONFIG : 'F U T, 0, 0, 0',
	X =   389.566  mm,	Y =     0.000  mm,	Z =     0.000  mm,
	W =  -167.363 deg,	P =     0.000 deg,	R =   105.687 deg
};
P[66]{
   GP1:
	UF : 7, UT : 3,	CONFIG : 'F U T, 0, 0, 0',
	X =   389.566  mm,	Y =     0.000  mm,	Z =     0.000  mm,
	W =  -167.363 deg,	P =     0.000 deg,	R =   105.687 deg
};
P[67]{
   GP1:
	UF : 7, UT : 3,	CONFIG : 'F U T, 0, 0, 0',
	X =   388.521  mm,	Y =    28.251  mm,	Z =     0.000  mm,
	W =  -167.364 deg,	P =     0.000 deg,	R =   109.338 deg
};
P[68]{
   GP1:
	UF : 7, UT : 3,	CONFIG : 'F U T, 0, 0, 0',
	X =   385.912  mm,	Y =    53.119  mm,	Z =     0.000  mm,
	W =  -167.363 deg,	P =     0.000 deg,	R =   112.986 deg
};
P[69]{
   GP1:
	UF : 7, UT : 3,	CONFIG : 'F U T, 0, 0, 0',
	X =   381.670  mm,	Y =    77.969  mm,	Z =     0.000  mm,
	W =  -167.363 deg,	P =     0.001 deg,	R =   116.656 deg
};
P[70]{
   GP1:
	UF : 7, UT : 3,	CONFIG : 'F U T, 0, 0, 0',
	X =   375.876  mm,	Y =   102.316  mm,	Z =     0.000  mm,
	W =  -167.363 deg,	P =     0.001 deg,	R =   120.286 deg
};
P[71]{
   GP1:
	UF : 7, UT : 3,	CONFIG : 'F U T, 0, 0, 0',
	X =   368.481  mm,	Y =   126.382  mm,	Z =     0.000  mm,
	W =  -167.363 deg,	P =     0.001 deg,	R =   123.955 deg
};
P[72]{
   GP1:
	UF : 7, UT : 3,	CONFIG : 'F U T, 0, 0, 0',
	X =   359.567  mm,	Y =   149.869  mm,	Z =     0.000  mm,
	W =  -167.363 deg,	P =     0.001 deg,	R =   127.612 deg
};
P[73]{
   GP1:
	UF : 7, UT : 3,	CONFIG : 'F U T, 0, 0, 0',
	X =   349.134  mm,	Y =   172.780  mm,	Z =     0.000  mm,
	W =  -167.363 deg,	P =     0.001 deg,	R =   131.276 deg
};
P[74]{
   GP1:
	UF : 7, UT : 3,	CONFIG : 'F U T, 0, 0, 0',
	X =   337.372  mm,	Y =   194.743  mm,	Z =     0.000  mm,
	W =  -167.363 deg,	P =     0.002 deg,	R =   134.933 deg
};
P[75]{
   GP1:
	UF : 7, UT : 3,	CONFIG : 'F U T, 0, 0, 0',
	X =   324.506  mm,	Y =   215.499  mm,	Z =     0.000  mm,
	W =  -167.363 deg,	P =     0.002 deg,	R =   138.631 deg
};
P[76]{
   GP1:
	UF : 7, UT : 3,	CONFIG : 'F U T, 0, 0, 0',
	X =   310.187  mm,	Y =   235.649  mm,	Z =     0.000  mm,
	W =  -167.362 deg,	P =     0.002 deg,	R =   142.292 deg
};
P[77]{
   GP1:
	UF : 7, UT : 3,	CONFIG : 'F U T, 0, 0, 0',
	X =   294.671  mm,	Y =   254.793  mm,	Z =     0.000  mm,
	W =  -167.362 deg,	P =     0.002 deg,	R =   145.974 deg
};
P[78]{
   GP1:
	UF : 7, UT : 3,	CONFIG : 'F U T, 0, 0, 0',
	X =   277.720  mm,	Y =   273.182  mm,	Z =     0.000  mm,
	W =  -167.362 deg,	P =     0.002 deg,	R =   149.643 deg
};
P[79]{
   GP1:
	UF : 7, UT : 3,	CONFIG : 'F U T, 0, 0, 0',
	X =   259.651  mm,	Y =   290.406  mm,	Z =     0.000  mm,
	W =  -167.361 deg,	P =     0.002 deg,	R =   153.265 deg
};
P[80]{
   GP1:
	UF : 7, UT : 3,	CONFIG : 'F U T, 0, 0, 0',
	X =   240.452  mm,	Y =   306.492  mm,	Z =     0.000  mm,
	W =  -167.361 deg,	P =     0.002 deg,	R =   156.913 deg
};
P[81]{
   GP1:
	UF : 7, UT : 3,	CONFIG : 'F U T, 0, 0, 0',
	X =   220.362  mm,	Y =   321.235  mm,	Z =     0.000  mm,
	W =  -167.361 deg,	P =     0.002 deg,	R =   160.552 deg
};
P[82]{
   GP1:
	UF : 7, UT : 3,	CONFIG : 'F U T, 0, 0, 0',
	X =   199.383  mm,	Y =   334.655  mm,	Z =     0.000  mm,
	W =  -167.361 deg,	P =     0.002 deg,	R =   164.192 deg
};
P[83]{
   GP1:
	UF : 7, UT : 3,	CONFIG : 'F U T, 0, 0, 0',
	X =   177.682  mm,	Y =   346.659  mm,	Z =     0.000  mm,
	W =  -167.360 deg,	P =     0.002 deg,	R =   167.858 deg
};
P[84]{
   GP1:
	UF : 7, UT : 3,	CONFIG : 'F U T, 0, 0, 0',
	X =   155.292  mm,	Y =   357.250  mm,	Z =     0.000  mm,
	W =  -167.360 deg,	P =     0.002 deg,	R =   171.541 deg
};
P[85]{
   GP1:
	UF : 7, UT : 3,	CONFIG : 'F U T, 0, 0, 0',
	X =   132.407  mm,	Y =   366.355  mm,	Z =     0.000  mm,
	W =  -167.360 deg,	P =     0.002 deg,	R =   175.213 deg
};
P[86]{
   GP1:
	UF : 7, UT : 3,	CONFIG : 'F U T, 0, 0, 0',
	X =   108.756  mm,	Y =   374.064  mm,	Z =     0.000  mm,
	W =  -167.359 deg,	P =     0.002 deg,	R =   178.880 deg
};
P[87]{
   GP1:
	UF : 7, UT : 3,	CONFIG : 'F U T, 0, 0, 0',
	X =    84.546  mm,	Y =   380.276  mm,	Z =     0.000  mm,
	W =  -167.359 deg,	P =     0.002 deg,	R =  -177.447 deg
};
P[88]{
   GP1:
	UF : 7, UT : 3,	CONFIG : 'F U T, 0, 0, 0',
	X =    59.937  mm,	Y =   384.926  mm,	Z =     0.000  mm,
	W =  -167.359 deg,	P =     0.001 deg,	R =  -173.789 deg
};
P[89]{
   GP1:
	UF : 7, UT : 3,	CONFIG : 'F U T, 0, 0, 0',
	X =    35.074  mm,	Y =   387.979  mm,	Z =     0.000  mm,
	W =  -167.358 deg,	P =     0.001 deg,	R =  -170.140 deg
};
P[90]{
   GP1:
	UF : 7, UT : 3,	CONFIG : 'F U T, 0, 0, 0',
	X =    10.231  mm,	Y =   389.420  mm,	Z =     0.000  mm,
	W =  -167.358 deg,	P =     0.001 deg,	R =  -166.491 deg
};
P[91]{
   GP1:
